LIN {X 0,Y 446.411,Z 696.876,A -85,B 0,C 180,E1 -8692.12,E2 -8692.12} C_VEL
LIN {X 0,Y 446.428,Z 696.878,A -85,B 0,C 180,E1 -8695.476,E2 -8695.476} C_VEL
LIN {X 0,Y 446.472,Z 697.063,A -85,B 0,C 180,E1 -8698.506,E2 -8698.506} C_VEL
LIN {X 0,Y 449.672,Z 710.867,A -85,B 0,C 180,E1 -8700.763,E2 -8700.763} C_VEL
LIN {X 0,Y 451.142,Z 718.019,A -85,B 0,C 180,E1 -8701.884,E2 -8701.884} C_VEL
LIN {X 0,Y 450.044,Z 738.904,A -85,B 0,C 180,E1 -8704.839,E2 -8704.839} C_VEL
LIN {X 0,Y 448.95,Z 761.08,A -85,B 0,C 180,E1 -8707.931,E2 -8707.931} C_VEL
LIN {X 0,Y 447.767,Z 788.534,A -85,B 0,C 180,E1 -8711.704,E2 -8711.704} C_VEL
LIN {X 0,Y 447.645,Z 792.086,A -85,B 0,C 180,E1 -8712.146,E2 -8712.146} C_VEL
LIN {X 0,Y 450.644,Z 820.359,A -85,B 0,C 180,E1 -8712.733,E2 -8712.733} C_VEL
LIN {X 0,Y 449.869,Z 902.501,A -85,B 0,C 180,E1 -8714.074,E2 -8714.074} C_VEL
LIN {X 0,Y 449.392,Z 915.74,A -85,B 0,C 180,E1 -8714.464,E2 -8714.464} C_VEL
LIN {X 0,Y 448.928,Z 927.38,A -85,B 0,C 180,E1 -8714.971,E2 -8714.971} C_VEL
LIN {X 0,Y 448.223,Z 939.892,A -85,B 0,C 180,E1 -8715.701,E2 -8715.701} C_VEL
LIN {X 0,Y 447.645,Z 951.783,A -85,B 0,C 180,E1 -8716.617,E2 -8716.617} C_VEL
LIN {X 0,Y 447.169,Z 962.339,A -85,B 0,C 180,E1 -8717.634,E2 -8717.634} C_VEL
LIN {X 0,Y 446.635,Z 971.045,A -85,B 0,C 180,E1 -8718.655,E2 -8718.655} C_VEL
LIN {X 0,Y 446.239,Z 979.102,A -85,B 0,C 180,E1 -8719.793,E2 -8719.793} C_VEL
LIN {X 0,Y 445.972,Z 987.009,A -85,B 0,C 180,E1 -8721.16,E2 -8721.16} C_VEL
LIN {X 0,Y 445.778,Z 994.294,A -85,B 0,C 180,E1 -8722.753,E2 -8722.753} C_VEL
LIN {X 0,Y 445.753,Z 999.161,A -85,B 0,C 180,E1 -8724.117,E2 -8724.117} C_VEL
LIN {X 0,Y 445.749,Z 1002.881,A -85,B 0,C 180,E1 -8725.477,E2 -8725.477} C_VEL
LIN {X 0,Y 445.775,Z 1004.802,A -85,B 0,C 180,E1 -8726.383,E2 -8726.383} C_VEL
LIN {X 0,Y 445.737,Z 1006.233,A -85,B 0,C 180,E1 -8727.287,E2 -8727.287} C_VEL
LIN {X 0,Y 445.739,Z 1007.252,A -85,B 0,C 180,E1 -8728.192,E2 -8728.192} C_VEL
LIN {X 0,Y 445.731,Z 1007.867,A -85,B 0,C 180,E1 -8729.095,E2 -8729.095} C_VEL
LIN {X 0,Y 445.738,Z 1008.078,A -85,B 0,C 180,E1 -8729.999,E2 -8729.999} C_VEL
LIN {X 0,Y 445.735,Z 1007.841,A -85,B 0,C 180,E1 -8730.902,E2 -8730.902} C_VEL
LIN {X 0,Y 445.746,Z 1007.198,A -85,B 0,C 180,E1 -8731.806,E2 -8731.806} C_VEL
LIN {X 0,Y 445.745,Z 1006.152,A -85,B 0,C 180,E1 -8732.71,E2 -8732.71} C_VEL
LIN {X 0,Y 445.774,Z 1004.693,A -85,B 0,C 180,E1 -8733.614,E2 -8733.614} C_VEL
LIN {X 0,Y 445.767,Z 1001.629,A -85,B 0,C 180,E1 -8734.973,E2 -8734.973} C_VEL
LIN {X 0,Y 445.748,Z 996.417,A -85,B 0,C 180,E1 -8736.632,E2 -8736.632} C_VEL
LIN {X 0,Y 445.887,Z 990.109,A -85,B 0,C 180,E1 -8738.154,E2 -8738.154} C_VEL
LIN {X 0,Y 446.086,Z 982.981,A -85,B 0,C 180,E1 -8739.521,E2 -8739.521} C_VEL
LIN {X 0,Y 446.484,Z 974.101,A -85,B 0,C 180,E1 -8740.887,E2 -8740.887} C_VEL
LIN {X 0,Y 446.893,Z 965.022,A -85,B 0,C 180,E1 -8742.026,E2 -8742.026} C_VEL
LIN {X 0,Y 447.39,Z 956.062,A -85,B 0,C 180,E1 -8742.956,E2 -8742.956} C_VEL
LIN {X 0,Y 447.891,Z 944.244,A -85,B 0,C 180,E1 -8743.959,E2 -8743.959} C_VEL
LIN {X 0,Y 448.619,Z 932.176,A -85,B 0,C 180,E1 -8744.747,E2 -8744.747} C_VEL
LIN {X 0,Y 449.176,Z 919.643,A -85,B 0,C 180,E1 -8745.366,E2 -8745.366} C_VEL
LIN {X 0,Y 449.722,Z 906.777,A -85,B 0,C 180,E1 -8745.812,E2 -8745.812} C_VEL
LIN {X 0,Y 449.986,Z 891.416,A -85,B 0,C 180,E1 -8746.122,E2 -8746.122} C_VEL
LIN {X 0,Y 450.614,Z 818.515,A -85,B 0,C 180,E1 -8747.294,E2 -8747.294} C_VEL
LIN {X 0,Y 447.578,Z 790.826,A -85,B 0,C 180,E1 -8747.892,E2 -8747.892} C_VEL
LIN {X 0,Y 448.442,Z 768.678,A -85,B 0,C 180,E1 -8750.886,E2 -8750.886} C_VEL
LIN {X 0,Y 449.417,Z 748.03,A -85,B 0,C 180,E1 -8753.744,E2 -8753.744} C_VEL
LIN {X 0,Y 450.55,Z 725.648,A -85,B 0,C 180,E1 -8756.894,E2 -8756.894} C_VEL
LIN {X 0,Y 450.925,Z 717.026,A -85,B 0,C 180,E1 -8758.128,E2 -8758.128} C_VEL
LIN {X 0,Y 447.652,Z 702.006,A -85,B 0,C 180,E1 -8760.532,E2 -8760.532} C_VEL
LIN {X 0,Y 446.437,Z 696.965,A -85,B 0,C 180,E1 -8761.428,E2 -8761.428} C_VEL
LIN {X 0,Y 446.423,Z 696.872,A -85,B 0,C 180,E1 -8764.522,E2 -8764.522} C_VEL
LIN {X 0,Y 446.409,Z 696.878,A -85,B 0,C 180,E1 -8768.078,E2 -8768.078} C_VEL
LIN {X 0,Y 446.42,Z 696.878,A -85,B 0,C 180,E1 -8770.916,E2 -8770.916} C_VEL
LIN {X 0,Y 446.394,Z 696.876,A -85,B 0,C 180,E1 -8773.845,E2 -8773.845} C_VEL
LIN {X 0,Y 446.415,Z 696.873,A -85,B 0,C 180,E1 -8776.399,E2 -8776.399} C_VEL
LIN {X 0,Y 446.439,Z 696.864,A -85,B 0,C 180,E1 -8779.802,E2 -8779.802} C_VEL
LIN {X 0,Y 446.418,Z 696.874,A -85,B 0,C 180,E1 -8782.122,E2 -8782.122} C_VEL
LIN {X 0,Y 446.421,Z 696.874,A -85,B 0,C 180,E1 -8785.476,E2 -8785.476} C_VEL
LIN {X 0,Y 446.409,Z 696.876,A -85,B 0,C 180,E1 -8788.699,E2 -8788.699} C_VEL
LIN {X 0,Y 446.473,Z 696.867,A -85,B 0,C 180,E1 -8791.821,E2 -8791.821} C_VEL
LIN {X 0,Y 446.447,Z 696.87,A -85,B 0,C 180,E1 -8794.847,E2 -8794.847} C_VEL
LIN {X 0,Y 446.436,Z 696.868,A -85,B 0,C 180,E1 -8798.244,E2 -8798.244} C_VEL
LIN {X 0,Y 446.446,Z 696.874,A -85,B 0,C 180,E1 -8801.649,E2 -8801.649} C_VEL
LIN {X 0,Y 446.504,Z 696.863,A -85,B 0,C 180,E1 -8804.48,E2 -8804.48} C_VEL
LIN {X 0,Y 446.505,Z 696.867,A -85,B 0,C 180,E1 -8808.193,E2 -8808.193} C_VEL
LIN {X 0,Y 446.588,Z 696.851,A -85,B 0,C 180,E1 -8811.858,E2 -8811.858} C_VEL
LIN {X 0,Y 446.63,Z 696.846,A -85,B 0,C 180,E1 -8814.583,E2 -8814.583} C_VEL
LIN {X 0,Y 446.698,Z 696.837,A -85,B 0,C 180,E1 -8817.295,E2 -8817.295} C_VEL
LIN {X 0,Y 446.78,Z 696.829,A -85,B 0,C 180,E1 -8820,E2 -8820} C_VEL
LIN {X 0,Y 446.696,Z 696.842,A -85,B 0,C 180,E1 -8822.706,E2 -8822.706} C_VEL
LIN {X 0,Y 446.627,Z 696.851,A -85,B 0,C 180,E1 -8826.324,E2 -8826.324} C_VEL
LIN {X 0,Y 446.527,Z 696.862,A -85,B 0,C 180,E1 -8829.056,E2 -8829.056} C_VEL
LIN {X 0,Y 446.509,Z 696.864,A -85,B 0,C 180,E1 -8832.73,E2 -8832.73} C_VEL
LIN {X 0,Y 446.484,Z 696.862,A -85,B 0,C 180,E1 -8836.228,E2 -8836.228} C_VEL
LIN {X 0,Y 446.457,Z 696.872,A -85,B 0,C 180,E1 -8839.304,E2 -8839.304} C_VEL
LIN {X 0,Y 446.406,Z 696.872,A -85,B 0,C 180,E1 -8842.2,E2 -8842.2} C_VEL
LIN {X 0,Y 446.428,Z 696.873,A -85,B 0,C 180,E1 -8845.154,E2 -8845.154} C_VEL
LIN {X 0,Y 446.475,Z 696.86,A -85,B 0,C 180,E1 -8848.18,E2 -8848.18} C_VEL
LIN {X 0,Y 446.41,Z 696.875,A -85,B 0,C 180,E1 -8851.776,E2 -8851.776} C_VEL
LIN {X 0,Y 446.421,Z 696.874,A -85,B 0,C 180,E1 -8854.524,E2 -8854.524} C_VEL
LIN {X 0,Y 446.422,Z 696.874,A -85,B 0,C 180,E1 -8858.083,E2 -8858.083} C_VEL
LIN {X 0,Y 446.419,Z 696.874,A -85,B 0,C 180,E1 -8860.919,E2 -8860.919} C_VEL
LIN {X 0,Y 446.393,Z 696.883,A -85,B 0,C 180,E1 -8863.847,E2 -8863.847} C_VEL
LIN {X 0,Y 446.424,Z 696.869,A -85,B 0,C 180,E1 -8866.781,E2 -8866.781} C_VEL
LIN {X 0,Y 446.468,Z 697.125,A -85,B 0,C 180,E1 -8867.456,E2 -8867.456} C_VEL
LIN {X 0,Y 446.776,Z 698.3,A -85,B 0,C 180,E1 -8867.596,E2 -8867.596} C_VEL
LIN {X 0,Y 451.11,Z 709.604,A -85,B 0,C 180,E1 -8867.983,E2 -8867.983} C_VEL
LIN {X 0,Y 450.672,Z 778.842,A -85,B 0,C 180,E1 -8869.143,E2 -8869.143} C_VEL
LIN {X 0,Y 450.538,Z 792.347,A -85,B 0,C 180,E1 -8869.566,E2 -8869.566} C_VEL
LIN {X 0,Y 450.352,Z 805.1,A -85,B 0,C 180,E1 -8870.162,E2 -8870.162} C_VEL
LIN {X 0,Y 450.013,Z 816.865,A -85,B 0,C 180,E1 -8870.911,E2 -8870.911} C_VEL
LIN {X 0,Y 449.474,Z 828.486,A -85,B 0,C 180,E1 -8871.859,E2 -8871.859} C_VEL
LIN {X 0,Y 448.979,Z 838.696,A -85,B 0,C 180,E1 -8872.914,E2 -8872.914} C_VEL
LIN {X 0,Y 448.445,Z 847.302,A -85,B 0,C 180,E1 -8874.008,E2 -8874.008} C_VEL
LIN {X 0,Y 447.898,Z 855.784,A -85,B 0,C 180,E1 -8875.335,E2 -8875.335} C_VEL
LIN {X 0,Y 447.493,Z 862.578,A -85,B 0,C 180,E1 -8876.657,E2 -8876.657} C_VEL
LIN {X 0,Y 447.072,Z 868.448,A -85,B 0,C 180,E1 -8878.091,E2 -8878.091} C_VEL
LIN {X 0,Y 446.774,Z 873.624,A -85,B 0,C 180,E1 -8879.778,E2 -8879.778} C_VEL
LIN {X 0,Y 446.617,Z 876.016,A -85,B 0,C 180,E1 -8880.805,E2 -8880.805} C_VEL
LIN {X 0,Y 446.483,Z 877.801,A -85,B 0,C 180,E1 -8881.823,E2 -8881.823} C_VEL
LIN {X 0,Y 446.403,Z 879.102,A -85,B 0,C 180,E1 -8882.836,E2 -8882.836} C_VEL
LIN {X 0,Y 446.335,Z 879.859,A -85,B 0,C 180,E1 -8883.841,E2 -8883.841} C_VEL
LIN {X 0,Y 446.292,Z 880.159,A -85,B 0,C 180,E1 -8884.839,E2 -8884.839} C_VEL
LIN {X 0,Y 446.282,Z 879.919,A -85,B 0,C 180,E1 -8885.977,E2 -8885.977} C_VEL
LIN {X 0,Y 446.374,Z 878.253,A -85,B 0,C 180,E1 -8887.8,E2 -8887.8} C_VEL
LIN {X 0,Y 446.558,Z 875.728,A -85,B 0,C 180,E1 -8889.263,E2 -8889.263} C_VEL
LIN {X 0,Y 446.761,Z 872.127,A -85,B 0,C 180,E1 -8890.712,E2 -8890.712} C_VEL
LIN {X 0,Y 446.814,Z 871.213,A -85,B 0,C 180,E1 -8891.008,E2 -8891.008} C_VEL
LIN {X 0,Y 446.302,Z 869.052,A -85,B 0,C 180,E1 -8891.709,E2 -8891.709} C_VEL
LIN {X 0,Y 443.732,Z 865.275,A -85,B 0,C 180,E1 -8892.844,E2 -8892.844} C_VEL
LIN {X 0,Y 441.198,Z 860.875,A -85,B 0,C 180,E1 -8893.948,E2 -8893.948} C_VEL
LIN {X 0,Y 440.742,Z 857.682,A -85,B 0,C 180,E1 -8894.594,E2 -8894.594} C_VEL
LIN {X 0,Y 441.292,Z 849.452,A -85,B 0,C 180,E1 -8895.945,E2 -8895.945} C_VEL
LIN {X 0,Y 441.805,Z 840.503,A -85,B 0,C 180,E1 -8897.134,E2 -8897.134} C_VEL
LIN {X 0,Y 442.34,Z 830.654,A -85,B 0,C 180,E1 -8898.198,E2 -8898.198} C_VEL
LIN {X 0,Y 442.866,Z 819.969,A -85,B 0,C 180,E1 -8899.129,E2 -8899.129} C_VEL
LIN {X 0,Y 443.254,Z 807.77,A -85,B 0,C 180,E1 -8899.957,E2 -8899.957} C_VEL
LIN {X 0,Y 443.562,Z 795.192,A -85,B 0,C 180,E1 -8900.597,E2 -8900.597} C_VEL
LIN {X 0,Y 443.715,Z 782.628,A -85,B 0,C 180,E1 -8901.044,E2 -8901.044} C_VEL
LIN {X 0,Y 443.753,Z 767.637,A -85,B 0,C 180,E1 -8901.355,E2 -8901.355} C_VEL
LIN {X 0,Y 444.215,Z 710.877,A -85,B 0,C 180,E1 -8902.29,E2 -8902.29} C_VEL
LIN {X 0,Y 439.707,Z 698.68,A -85,B 0,C 180,E1 -8902.707,E2 -8902.707} C_VEL
LIN {X 0,Y 439.558,Z 697.817,A -85,B 0,C 180,E1 -8902.883,E2 -8902.883} C_VEL
LIN {X 0,Y 439.599,Z 697.729,A -85,B 0,C 180,E1 -8904.497,E2 -8904.497} C_VEL
LIN {X 0,Y 439.629,Z 697.724,A -85,B 0,C 180,E1 -8908.169,E2 -8908.169} C_VEL
LIN {X 0,Y 439.672,Z 697.718,A -85,B 0,C 180,E1 -8910.001,E2 -8910.001} C_VEL
LIN {X 0,Y 439.605,Z 697.727,A -85,B 0,C 180,E1 -8912.75,E2 -8912.75} C_VEL
LIN {X 0,Y 439.562,Z 697.732,A -85,B 0,C 180,E1 -8916.427,E2 -8916.427} C_VEL
LIN {X 0,Y 439.476,Z 697.739,A -85,B 0,C 180,E1 -8919.203,E2 -8919.203} C_VEL
LIN {X 0,Y 439.47,Z 697.742,A -85,B 0,C 180,E1 -8922.939,E2 -8922.939} C_VEL
LIN {X 0,Y 439.45,Z 697.741,A -85,B 0,C 180,E1 -8926.348,E2 -8926.348} C_VEL
LIN {X 0,Y 439.385,Z 697.741,A -85,B 0,C 180,E1 -8929.628,E2 -8929.628} C_VEL
LIN {X 0,Y 439.367,Z 697.754,A -85,B 0,C 180,E1 -8932.577,E2 -8932.577} C_VEL
LIN {X 0,Y 439.349,Z 697.746,A -85,B 0,C 180,E1 -8935.59,E2 -8935.59} C_VEL
LIN {X 0,Y 439.383,Z 697.747,A -85,B 0,C 180,E1 -8938.677,E2 -8938.677} C_VEL
LIN {X 0,Y 439.348,Z 697.751,A -85,B 0,C 180,E1 -8942.025,E2 -8942.025} C_VEL
LIN {X 0,Y 439.388,Z 697.737,A -85,B 0,C 180,E1 -8945.338,E2 -8945.338} C_VEL
LIN {X 0,Y 439.353,Z 697.752,A -85,B 0,C 180,E1 -8948.599,E2 -8948.599} C_VEL
LIN {X 0,Y 439.35,Z 697.754,A -85,B 0,C 180,E1 -8952.211,E2 -8952.211} C_VEL
LIN {X 0,Y 439.377,Z 697.754,A -85,B 0,C 180,E1 -8955.267,E2 -8955.267} C_VEL
LIN {X 0,Y 439.365,Z 697.752,A -85,B 0,C 180,E1 -8958.748,E2 -8958.748} C_VEL
LIN {X 0,Y 439.355,Z 697.759,A -85,B 0,C 180,E1 -8961.613,E2 -8961.613} C_VEL
LIN {X 0,Y 439.357,Z 697.755,A -85,B 0,C 180,E1 -8964.84,E2 -8964.84} C_VEL
LIN {X 0,Y 439.352,Z 697.76,A -85,B 0,C 180,E1 -8968.137,E2 -8968.137} C_VEL
LIN {X 0,Y 439.423,Z 697.912,A -85,B 0,C 180,E1 -8969.481,E2 -8969.481} C_VEL
LIN {X 0,Y 439.563,Z 698.75,A -85,B 0,C 180,E1 -8969.623,E2 -8969.623} C_VEL
LIN {X 0,Y 443.704,Z 710.36,A -85,B 0,C 180,E1 -8970.015,E2 -8970.015} C_VEL
LIN {X 0,Y 443.036,Z 773.791,A -85,B 0,C 180,E1 -8971.157,E2 -8971.157} C_VEL
LIN {X 0,Y 442.834,Z 785.481,A -85,B 0,C 180,E1 -8971.507,E2 -8971.507} C_VEL
LIN {X 0,Y 442.604,Z 795.704,A -85,B 0,C 180,E1 -8971.939,E2 -8971.939} C_VEL
LIN {X 0,Y 442.436,Z 804.955,A -85,B 0,C 180,E1 -8972.442,E2 -8972.442} C_VEL
LIN {X 0,Y 441.975,Z 815.897,A -85,B 0,C 180,E1 -8973.193,E2 -8973.193} C_VEL
LIN {X 0,Y 441.652,Z 824.568,A -85,B 0,C 180,E1 -8973.922,E2 -8973.922} C_VEL
LIN {X 0,Y 441.184,Z 832.911,A -85,B 0,C 180,E1 -8974.754,E2 -8974.754} C_VEL
LIN {X 0,Y 440.818,Z 841.284,A -85,B 0,C 180,E1 -8975.761,E2 -8975.761} C_VEL
LIN {X 0,Y 440.485,Z 848.193,A -85,B 0,C 180,E1 -8976.741,E2 -8976.741} C_VEL
LIN {X 0,Y 440.108,Z 854.791,A -85,B 0,C 180,E1 -8977.851,E2 -8977.851} C_VEL
LIN {X 0,Y 439.75,Z 861.198,A -85,B 0,C 180,E1 -8979.17,E2 -8979.17} C_VEL
LIN {X 0,Y 439.507,Z 866.87,A -85,B 0,C 180,E1 -8980.642,E2 -8980.642} C_VEL
LIN {X 0,Y 439.289,Z 870.516,A -85,B 0,C 180,E1 -8981.822,E2 -8981.822} C_VEL
LIN {X 0,Y 439.14,Z 873.848,A -85,B 0,C 180,E1 -8983.257,E2 -8983.257} C_VEL
LIN {X 0,Y 439.079,Z 875.563,A -85,B 0,C 180,E1 -8984.21,E2 -8984.21} C_VEL
LIN {X 0,Y 439.007,Z 877.457,A -85,B 0,C 180,E1 -8986.105,E2 -8986.105} C_VEL
LIN {X 0,Y 439.052,Z 877.759,A -85,B 0,C 180,E1 -8987.542,E2 -8987.542} C_VEL
LIN {X 0,Y 439.106,Z 877.048,A -85,B 0,C 180,E1 -8988.927,E2 -8988.927} C_VEL
LIN {X 0,Y 439.205,Z 876.169,A -85,B 0,C 180,E1 -8989.862,E2 -8989.862} C_VEL
LIN {X 0,Y 439.405,Z 872.864,A -85,B 0,C 180,E1 -8991.723,E2 -8991.723} C_VEL
LIN {X 0,Y 439.571,Z 870.661,A -85,B 0,C 180,E1 -8992.651,E2 -8992.651} C_VEL
LIN {X 0,Y 439.83,Z 866.295,A -85,B 0,C 180,E1 -8994.038,E2 -8994.038} C_VEL
LIN {X 0,Y 440.123,Z 860.682,A -85,B 0,C 180,E1 -8995.42,E2 -8995.42} C_VEL
LIN {X 0,Y 440.456,Z 854.971,A -85,B 0,C 180,E1 -8996.569,E2 -8996.569} C_VEL
LIN {X 0,Y 440.907,Z 848.065,A -85,B 0,C 180,E1 -8997.716,E2 -8997.716} C_VEL
LIN {X 0,Y 441.349,Z 839.698,A -85,B 0,C 180,E1 -8998.859,E2 -8998.859} C_VEL
LIN {X 0,Y 441.764,Z 831.673,A -85,B 0,C 180,E1 -8999.772,E2 -8999.772} C_VEL
LIN {X 0,Y 442.208,Z 823.29,A -85,B 0,C 180,E1 -9000.569,E2 -9000.569} C_VEL
LIN {X 0,Y 442.55,Z 814.752,A -85,B 0,C 180,E1 -9001.251,E2 -9001.251} C_VEL
LIN {X 0,Y 442.87,Z 804.092,A -85,B 0,C 180,E1 -9001.932,E2 -9001.932} C_VEL
LIN {X 0,Y 443.183,Z 793.086,A -85,B 0,C 180,E1 -9002.471,E2 -9002.471} C_VEL
LIN {X 0,Y 443.272,Z 782.09,A -85,B 0,C 180,E1 -9002.868,E2 -9002.868} C_VEL
LIN {X 0,Y 443.347,Z 770.375,A -85,B 0,C 180,E1 -9003.152,E2 -9003.152} C_VEL
LIN {X 0,Y 444.19,Z 710.257,A -85,B 0,C 180,E1 -9004.252,E2 -9004.252} C_VEL
LIN {X 0,Y 439.633,Z 698.633,A -85,B 0,C 180,E1 -9004.728,E2 -9004.728} C_VEL
LIN {X 0,Y 439.496,Z 697.795,A -85,B 0,C 180,E1 -9004.931,E2 -9004.931} C_VEL
LIN {X 0,Y 439.56,Z 697.732,A -85,B 0,C 180,E1 -9007.556,E2 -9007.556} C_VEL
LIN {X 0,Y 439.467,Z 697.744,A -85,B 0,C 180,E1 -9010.132,E2 -9010.132} C_VEL
LIN {X 0,Y 439.473,Z 697.741,A -85,B 0,C 180,E1 -9012.937,E2 -9012.937} C_VEL
LIN {X 0,Y 439.454,Z 697.747,A -85,B 0,C 180,E1 -9016.348,E2 -9016.348} C_VEL
LIN {X 0,Y 439.409,Z 697.748,A -85,B 0,C 180,E1 -9019.626,E2 -9019.626} C_VEL
LIN {X 0,Y 439.371,Z 697.758,A -85,B 0,C 180,E1 -9022.575,E2 -9022.575} C_VEL
LIN {X 0,Y 439.387,Z 697.751,A -85,B 0,C 180,E1 -9025.586,E2 -9025.586} C_VEL
LIN {X 0,Y 439.407,Z 697.752,A -85,B 0,C 180,E1 -9028.674,E2 -9028.674} C_VEL
LIN {X 0,Y 439.375,Z 697.752,A -85,B 0,C 180,E1 -9032.029,E2 -9032.029} C_VEL
LIN {X 0,Y 439.399,Z 697.753,A -85,B 0,C 180,E1 -9035.339,E2 -9035.339} C_VEL
LIN {X 0,Y 439.39,Z 697.752,A -85,B 0,C 180,E1 -9038.594,E2 -9038.594} C_VEL
LIN {X 0,Y 439.395,Z 697.753,A -85,B 0,C 180,E1 -9041.256,E2 -9041.256} C_VEL
LIN {X 0,Y 439.406,Z 697.75,A -85,B 0,C 180,E1 -9044.729,E2 -9044.729} C_VEL
LIN {X 0,Y 439.402,Z 697.752,A -85,B 0,C 180,E1 -9047.795,E2 -9047.795} C_VEL
LIN {X 0,Y 439.395,Z 697.749,A -85,B 0,C 180,E1 -9050.222,E2 -9050.222} C_VEL
LIN {X 0,Y 439.377,Z 697.756,A -85,B 0,C 180,E1 -9053.712,E2 -9053.712} C_VEL
LIN {X 0,Y 439.377,Z 697.755,A -85,B 0,C 180,E1 -9057.053,E2 -9057.053} C_VEL
LIN {X 0,Y 439.432,Z 698.009,A -85,B 0,C 180,E1 -9058.244,E2 -9058.244} C_VEL
LIN {X 0,Y 442.655,Z 711.641,A -85,B 0,C 180,E1 -9060.514,E2 -9060.514} C_VEL
LIN {X 0,Y 444.151,Z 718.815,A -85,B 0,C 180,E1 -9061.659,E2 -9061.659} C_VEL
LIN {X 0,Y 444.197,Z 722.176,A -85,B 0,C 180,E1 -9062.158,E2 -9062.158} C_VEL
LIN {X 0,Y 442.914,Z 742.94,A -85,B 0,C 180,E1 -9065.135,E2 -9065.135} C_VEL
LIN {X 0,Y 441.853,Z 763.539,A -85,B 0,C 180,E1 -9068.049,E2 -9068.049} C_VEL
LIN {X 0,Y 440.712,Z 789.399,A -85,B 0,C 180,E1 -9071.665,E2 -9071.665} C_VEL
LIN {X 0,Y 440.678,Z 790.898,A -85,B 0,C 180,E1 -9071.849,E2 -9071.849} C_VEL
LIN {X 0,Y 443.816,Z 820.934,A -85,B 0,C 180,E1 -9072.489,E2 -9072.489} C_VEL
LIN {X 0,Y 443.053,Z 901.376,A -85,B 0,C 180,E1 -9073.823,E2 -9073.823} C_VEL
LIN {X 0,Y 442.51,Z 914.65,A -85,B 0,C 180,E1 -9074.217,E2 -9074.217} C_VEL
LIN {X 0,Y 441.975,Z 927.448,A -85,B 0,C 180,E1 -9074.788,E2 -9074.788} C_VEL
LIN {X 0,Y 441.297,Z 938.844,A -85,B 0,C 180,E1 -9075.472,E2 -9075.472} C_VEL
LIN {X 0,Y 440.68,Z 950.445,A -85,B 0,C 180,E1 -9076.375,E2 -9076.375} C_VEL
LIN {X 0,Y 440.189,Z 961.306,A -85,B 0,C 180,E1 -9077.434,E2 -9077.434} C_VEL
LIN {X 0,Y 439.605,Z 970.012,A -85,B 0,C 180,E1 -9078.471,E2 -9078.471} C_VEL
LIN {X 0,Y 439.208,Z 978.077,A -85,B 0,C 180,E1 -9079.628,E2 -9079.628} C_VEL
LIN {X 0,Y 438.894,Z 985.985,A -85,B 0,C 180,E1 -9081.017,E2 -9081.017} C_VEL
LIN {X 0,Y 438.735,Z 993.279,A -85,B 0,C 180,E1 -9082.636,E2 -9082.636} C_VEL
LIN {X 0,Y 438.695,Z 998.148,A -85,B 0,C 180,E1 -9084.022,E2 -9084.022} C_VEL
LIN {X 0,Y 438.709,Z 1001.873,A -85,B 0,C 180,E1 -9085.404,E2 -9085.404} C_VEL
LIN {X 0,Y 438.736,Z 1003.795,A -85,B 0,C 180,E1 -9086.325,E2 -9086.325} C_VEL
LIN {X 0,Y 438.697,Z 1005.228,A -85,B 0,C 180,E1 -9087.244,E2 -9087.244} C_VEL
LIN {X 0,Y 438.702,Z 1006.247,A -85,B 0,C 180,E1 -9088.163,E2 -9088.163} C_VEL
LIN {X 0,Y 438.7,Z 1006.861,A -85,B 0,C 180,E1 -9089.081,E2 -9089.081} C_VEL
LIN {X 0,Y 438.71,Z 1007.072,A -85,B 0,C 180,E1 -9089.999,E2 -9089.999} C_VEL
LIN {X 0,Y 438.704,Z 1006.833,A -85,B 0,C 180,E1 -9090.917,E2 -9090.917} C_VEL
LIN {X 0,Y 438.71,Z 1006.188,A -85,B 0,C 180,E1 -9091.835,E2 -9091.835} C_VEL
LIN {X 0,Y 438.704,Z 1005.138,A -85,B 0,C 180,E1 -9092.753,E2 -9092.753} C_VEL
LIN {X 0,Y 438.736,Z 1003.677,A -85,B 0,C 180,E1 -9093.672,E2 -9093.672} C_VEL
LIN {X 0,Y 438.723,Z 1000.607,A -85,B 0,C 180,E1 -9095.053,E2 -9095.053} C_VEL
LIN {X 0,Y 438.684,Z 995.728,A -85,B 0,C 180,E1 -9096.645,E2 -9096.645} C_VEL
LIN {X 0,Y 438.849,Z 989.073,A -85,B 0,C 180,E1 -9098.286,E2 -9098.286} C_VEL
LIN {X 0,Y 439.036,Z 981.936,A -85,B 0,C 180,E1 -9099.675,E2 -9099.675} C_VEL
LIN {X 0,Y 439.426,Z 973.047,A -85,B 0,C 180,E1 -9101.064,E2 -9101.064} C_VEL
LIN {X 0,Y 439.922,Z 963.973,A -85,B 0,C 180,E1 -9102.219,E2 -9102.219} C_VEL
LIN {X 0,Y 440.479,Z 953.239,A -85,B 0,C 180,E1 -9103.336,E2 -9103.336} C_VEL
LIN {X 0,Y 441.036,Z 941.614,A -85,B 0,C 180,E1 -9104.298,E2 -9104.298} C_VEL
LIN {X 0,Y 441.86,Z 929.134,A -85,B 0,C 180,E1 -9105.095,E2 -9105.095} C_VEL
LIN {X 0,Y 442.377,Z 917.318,A -85,B 0,C 180,E1 -9105.667,E2 -9105.667} C_VEL
LIN {X 0,Y 442.872,Z 904.71,A -85,B 0,C 180,E1 -9106.092,E2 -9106.092} C_VEL
LIN {X 0,Y 443.154,Z 888.772,A -85,B 0,C 180,E1 -9106.407,E2 -9106.407} C_VEL
LIN {X 0,Y 443.713,Z 818.543,A -85,B 0,C 180,E1 -9107.559,E2 -9107.559} C_VEL
LIN {X 0,Y 440.628,Z 789.544,A -85,B 0,C 180,E1 -9108.204,E2 -9108.204} C_VEL
LIN {X 0,Y 441.791,Z 762.525,A -85,B 0,C 180,E1 -9111.951,E2 -9111.951} C_VEL
LIN {X 0,Y 442.938,Z 740.095,A -85,B 0,C 180,E1 -9115.13,E2 -9115.13} C_VEL
LIN {X 0,Y 444.111,Z 719.45,A -85,B 0,C 180,E1 -9118.107,E2 -9118.107} C_VEL
LIN {X 0,Y 441.632,Z 707.191,A -85,B 0,C 180,E1 -9120.083,E2 -9120.083} C_VEL
LIN {X 0,Y 439.387,Z 697.884,A -85,B 0,C 180,E1 -9121.689,E2 -9121.689} C_VEL
LIN {X 0,Y 439.381,Z 697.746,A -85,B 0,C 180,E1 -9124.042,E2 -9124.042} C_VEL
LIN {X 0,Y 439.342,Z 697.761,A -85,B 0,C 180,E1 -9126.886,E2 -9126.886} C_VEL
LIN {X 0,Y 439.394,Z 697.751,A -85,B 0,C 180,E1 -9129.848,E2 -9129.848} C_VEL
LIN {X 0,Y 439.374,Z 697.753,A -85,B 0,C 180,E1 -9132.626,E2 -9132.626} C_VEL
LIN {X 0,Y 439.398,Z 697.748,A -85,B 0,C 180,E1 -9135.27,E2 -9135.27} C_VEL
LIN {X 0,Y 439.381,Z 697.755,A -85,B 0,C 180,E1 -9138.742,E2 -9138.742} C_VEL
LIN {X 0,Y 439.375,Z 697.753,A -85,B 0,C 180,E1 -9141.605,E2 -9141.605} C_VEL
LIN {X 0,Y 439.391,Z 697.744,A -85,B 0,C 180,E1 -9144.843,E2 -9144.843} C_VEL
LIN {X 0,Y 439.364,Z 697.752,A -85,B 0,C 180,E1 -9148.139,E2 -9148.139} C_VEL
LIN {X 0,Y 439.414,Z 697.75,A -85,B 0,C 180,E1 -9151.326,E2 -9151.326} C_VEL
LIN {X 0,Y 439.394,Z 697.747,A -85,B 0,C 180,E1 -9154.414,E2 -9154.414} C_VEL
LIN {X 0,Y 439.354,Z 697.76,A -85,B 0,C 180,E1 -9157.424,E2 -9157.424} C_VEL
LIN {X 0,Y 439.429,Z 697.744,A -85,B 0,C 180,E1 -9160.662,E2 -9160.662} C_VEL
LIN {X 0,Y 439.463,Z 697.742,A -85,B 0,C 180,E1 -9164.225,E2 -9164.225} C_VEL
LIN {X 0,Y 439.471,Z 697.744,A -85,B 0,C 180,E1 -9168.001,E2 -9168.001} C_VEL
LIN {X 0,Y 439.536,Z 697.728,A -85,B 0,C 180,E1 -9171.726,E2 -9171.726} C_VEL
LIN {X 0,Y 439.605,Z 697.722,A -85,B 0,C 180,E1 -9174.496,E2 -9174.496} C_VEL
LIN {X 0,Y 439.624,Z 697.725,A -85,B 0,C 180,E1 -9178.168,E2 -9178.168} C_VEL
LIN {X 0,Y 439.751,Z 697.705,A -85,B 0,C 180,E1 -9180,E2 -9180} C_VEL
LIN {X 0,Y 439.643,Z 697.72,A -85,B 0,C 180,E1 -9182.749,E2 -9182.749} C_VEL
LIN {X 0,Y 439.601,Z 697.727,A -85,B 0,C 180,E1 -9186.426,E2 -9186.426} C_VEL
LIN {X 0,Y 439.489,Z 697.738,A -85,B 0,C 180,E1 -9189.202,E2 -9189.202} C_VEL
LIN {X 0,Y 439.453,Z 697.744,A -85,B 0,C 180,E1 -9192.938,E2 -9192.938} C_VEL
LIN {X 0,Y 439.435,Z 697.741,A -85,B 0,C 180,E1 -9196.349,E2 -9196.349} C_VEL
LIN {X 0,Y 439.391,Z 697.75,A -85,B 0,C 180,E1 -9199.627,E2 -9199.627} C_VEL
LIN {X 0,Y 439.352,Z 697.752,A -85,B 0,C 180,E1 -9202.576,E2 -9202.576} C_VEL
LIN {X 0,Y 439.377,Z 697.757,A -85,B 0,C 180,E1 -9205.587,E2 -9205.587} C_VEL
LIN {X 0,Y 439.407,Z 697.74,A -85,B 0,C 180,E1 -9208.675,E2 -9208.675} C_VEL
LIN {X 0,Y 439.361,Z 697.75,A -85,B 0,C 180,E1 -9212.032,E2 -9212.032} C_VEL
LIN {X 0,Y 439.387,Z 697.753,A -85,B 0,C 180,E1 -9215.342,E2 -9215.342} C_VEL
LIN {X 0,Y 439.382,Z 697.747,A -85,B 0,C 180,E1 -9218.596,E2 -9218.596} C_VEL
LIN {X 0,Y 439.381,Z 697.751,A -85,B 0,C 180,E1 -9221.258,E2 -9221.258} C_VEL
LIN {X 0,Y 439.392,Z 697.752,A -85,B 0,C 180,E1 -9224.731,E2 -9224.731} C_VEL
LIN {X 0,Y 439.396,Z 697.855,A -85,B 0,C 180,E1 -9227.096,E2 -9227.096} C_VEL
LIN {X 0,Y 439.574,Z 698.672,A -85,B 0,C 180,E1 -9227.262,E2 -9227.262} C_VEL
LIN {X 0,Y 444.534,Z 711.592,A -85,B 0,C 180,E1 -9227.732,E2 -9227.732} C_VEL
LIN {X 0,Y 443.906,Z 779.538,A -85,B 0,C 180,E1 -9228.882,E2 -9228.882} C_VEL
LIN {X 0,Y 443.782,Z 792.792,A -85,B 0,C 180,E1 -9229.297,E2 -9229.297} C_VEL
LIN {X 0,Y 443.601,Z 805.01,A -85,B 0,C 180,E1 -9229.865,E2 -9229.865} C_VEL
LIN {X 0,Y 443.328,Z 815.314,A -85,B 0,C 180,E1 -9230.501,E2 -9230.501} C_VEL
LIN {X 0,Y 442.818,Z 826.743,A -85,B 0,C 180,E1 -9231.397,E2 -9231.397} C_VEL
LIN {X 0,Y 442.311,Z 836.551,A -85,B 0,C 180,E1 -9232.363,E2 -9232.363} C_VEL
LIN {X 0,Y 441.719,Z 846.051,A -85,B 0,C 180,E1 -9233.514,E2 -9233.514} C_VEL
LIN {X 0,Y 441.143,Z 854.523,A -85,B 0,C 180,E1 -9234.778,E2 -9234.778} C_VEL
LIN {X 0,Y 440.687,Z 861.508,A -85,B 0,C 180,E1 -9236.072,E2 -9236.072} C_VEL
LIN {X 0,Y 440.26,Z 867.787,A -85,B 0,C 180,E1 -9237.526,E2 -9237.526} C_VEL
LIN {X 0,Y 439.84,Z 873.504,A -85,B 0,C 180,E1 -9239.25,E2 -9239.25} C_VEL
LIN {X 0,Y 439.607,Z 877.196,A -85,B 0,C 180,E1 -9240.819,E2 -9240.819} C_VEL
LIN {X 0,Y 439.431,Z 879.627,A -85,B 0,C 180,E1 -9242.369,E2 -9242.369} C_VEL
LIN {X 0,Y 439.344,Z 880.774,A -85,B 0,C 180,E1 -9243.613,E2 -9243.613} C_VEL
LIN {X 0,Y 439.265,Z 881.117,A -85,B 0,C 180,E1 -9245.42,E2 -9245.42} C_VEL
LIN {X 0,Y 439.258,Z 880.689,A -85,B 0,C 180,E1 -9246.424,E2 -9246.424} C_VEL
LIN {X 0,Y 439.393,Z 878.918,A -85,B 0,C 180,E1 -9248.08,E2 -9248.08} C_VEL
LIN {X 0,Y 439.639,Z 875.436,A -85,B 0,C 180,E1 -9249.899,E2 -9249.899} C_VEL
LIN {X 0,Y 439.881,Z 871.384,A -85,B 0,C 180,E1 -9251.366,E2 -9251.366} C_VEL
LIN {X 0,Y 440.237,Z 866.1,A -85,B 0,C 180,E1 -9252.824,E2 -9252.824} C_VEL
LIN {X 0,Y 440.64,Z 859.405,A -85,B 0,C 180,E1 -9254.269,E2 -9254.269} C_VEL
LIN {X 0,Y 440.742,Z 857.682,A -85,B 0,C 180,E1 -9254.594,E2 -9254.594} C_VEL
LIN {X 0,Y 440.292,Z 854.298,A -85,B 0,C 180,E1 -9255.224,E2 -9255.224} C_VEL
LIN {X 0,Y 437.825,Z 848.624,A -85,B 0,C 180,E1 -9256.241,E2 -9256.241} C_VEL
LIN {X 0,Y 435.444,Z 842.352,A -85,B 0,C 180,E1 -9257.198,E2 -9257.198} C_VEL
LIN {X 0,Y 435.117,Z 838.04,A -85,B 0,C 180,E1 -9257.725,E2 -9257.725} C_VEL
LIN {X 0,Y 435.696,Z 826.957,A -85,B 0,C 180,E1 -9258.841,E2 -9258.841} C_VEL
LIN {X 0,Y 436.214,Z 816.56,A -85,B 0,C 180,E1 -9259.674,E2 -9259.674} C_VEL
LIN {X 0,Y 436.576,Z 804.208,A -85,B 0,C 180,E1 -9260.446,E2 -9260.446} C_VEL
LIN {X 0,Y 436.822,Z 791.29,A -85,B 0,C 180,E1 -9261.035,E2 -9261.035} C_VEL
LIN {X 0,Y 436.958,Z 778.781,A -85,B 0,C 180,E1 -9261.416,E2 -9261.416} C_VEL
LIN {X 0,Y 437.466,Z 712.472,A -85,B 0,C 180,E1 -9262.544,E2 -9262.544} C_VEL
LIN {X 0,Y 432.708,Z 699.615,A -85,B 0,C 180,E1 -9262.992,E2 -9262.992} C_VEL
LIN {X 0,Y 432.533,Z 698.685,A -85,B 0,C 180,E1 -9263.184,E2 -9263.184} C_VEL
LIN {X 0,Y 432.574,Z 698.605,A -85,B 0,C 180,E1 -9264.407,E2 -9264.407} C_VEL
LIN {X 0,Y 432.599,Z 698.599,A -85,B 0,C 180,E1 -9268.139,E2 -9268.139} C_VEL
LIN {X 0,Y 432.623,Z 698.595,A -85,B 0,C 180,E1 -9270.001,E2 -9270.001} C_VEL
LIN {X 0,Y 432.558,Z 698.605,A -85,B 0,C 180,E1 -9272.795,E2 -9272.795} C_VEL
LIN {X 0,Y 432.519,Z 698.608,A -85,B 0,C 180,E1 -9276.532,E2 -9276.532} C_VEL
LIN {X 0,Y 432.422,Z 698.617,A -85,B 0,C 180,E1 -9279.355,E2 -9279.355} C_VEL
LIN {X 0,Y 432.436,Z 698.62,A -85,B 0,C 180,E1 -9282.804,E2 -9282.804} C_VEL
LIN {X 0,Y 432.416,Z 698.619,A -85,B 0,C 180,E1 -9286.478,E2 -9286.478} C_VEL
LIN {X 0,Y 432.322,Z 698.62,A -85,B 0,C 180,E1 -9289.963,E2 -9289.963} C_VEL
LIN {X 0,Y 432.315,Z 698.638,A -85,B 0,C 180,E1 -9292.966,E2 -9292.966} C_VEL
LIN {X 0,Y 432.301,Z 698.622,A -85,B 0,C 180,E1 -9296.038,E2 -9296.038} C_VEL
LIN {X 0,Y 432.321,Z 698.633,A -85,B 0,C 180,E1 -9299.19,E2 -9299.19} C_VEL
LIN {X 0,Y 432.311,Z 698.628,A -85,B 0,C 180,E1 -9302.445,E2 -9302.445} C_VEL
LIN {X 0,Y 432.336,Z 698.62,A -85,B 0,C 180,E1 -9305.819,E2 -9305.819} C_VEL
LIN {X 0,Y 432.317,Z 698.629,A -85,B 0,C 180,E1 -9308.71,E2 -9308.71} C_VEL
LIN {X 0,Y 432.306,Z 698.636,A -85,B 0,C 180,E1 -9311.802,E2 -9311.802} C_VEL
LIN {X 0,Y 432.317,Z 698.63,A -85,B 0,C 180,E1 -9314.351,E2 -9314.351} C_VEL
LIN {X 0,Y 432.306,Z 698.632,A -85,B 0,C 180,E1 -9317.019,E2 -9317.019} C_VEL
LIN {X 0,Y 432.294,Z 698.639,A -85,B 0,C 180,E1 -9319.829,E2 -9319.829} C_VEL
LIN {X 0,Y 432.293,Z 698.634,A -85,B 0,C 180,E1 -9323.02,E2 -9323.02} C_VEL
LIN {X 0,Y 432.327,Z 698.635,A -85,B 0,C 180,E1 -9326.005,E2 -9326.005} C_VEL
LIN {X 0,Y 432.377,Z 698.802,A -85,B 0,C 180,E1 -9329.229,E2 -9329.229} C_VEL
LIN {X 0,Y 432.617,Z 699.893,A -85,B 0,C 180,E1 -9329.387,E2 -9329.387} C_VEL
LIN {X 0,Y 436.893,Z 712.016,A -85,B 0,C 180,E1 -9329.79,E2 -9329.79} C_VEL
LIN {X 0,Y 436.19,Z 774.897,A -85,B 0,C 180,E1 -9330.946,E2 -9330.946} C_VEL
LIN {X 0,Y 435.974,Z 786.708,A -85,B 0,C 180,E1 -9331.309,E2 -9331.309} C_VEL
LIN {X 0,Y 435.73,Z 797.544,A -85,B 0,C 180,E1 -9331.784,E2 -9331.784} C_VEL
LIN {X 0,Y 435.517,Z 806.462,A -85,B 0,C 180,E1 -9332.284,E2 -9332.284} C_VEL
LIN {X 0,Y 435.1,Z 816.365,A -85,B 0,C 180,E1 -9332.971,E2 -9332.971} C_VEL
LIN {X 0,Y 434.739,Z 825.355,A -85,B 0,C 180,E1 -9333.733,E2 -9333.733} C_VEL
LIN {X 0,Y 434.232,Z 834.363,A -85,B 0,C 180,E1 -9334.653,E2 -9334.653} C_VEL
LIN {X 0,Y 433.881,Z 842.148,A -85,B 0,C 180,E1 -9335.603,E2 -9335.603} C_VEL
LIN {X 0,Y 433.542,Z 849.089,A -85,B 0,C 180,E1 -9336.599,E2 -9336.599} C_VEL
LIN {X 0,Y 433.119,Z 855.956,A -85,B 0,C 180,E1 -9337.775,E2 -9337.775} C_VEL
LIN {X 0,Y 432.782,Z 862.146,A -85,B 0,C 180,E1 -9339.068,E2 -9339.068} C_VEL
LIN {X 0,Y 432.516,Z 867.542,A -85,B 0,C 180,E1 -9340.47,E2 -9340.47} C_VEL
LIN {X 0,Y 432.338,Z 870.9,A -85,B 0,C 180,E1 -9341.519,E2 -9341.519} C_VEL
LIN {X 0,Y 432.148,Z 874.429,A -85,B 0,C 180,E1 -9342.978,E2 -9342.978} C_VEL
LIN {X 0,Y 432.097,Z 876.17,A -85,B 0,C 180,E1 -9343.948,E2 -9343.948} C_VEL
LIN {X 0,Y 431.999,Z 878.347,A -85,B 0,C 180,E1 -9345.875,E2 -9345.875} C_VEL
LIN {X 0,Y 432.042,Z 878.812,A -85,B 0,C 180,E1 -9347.43,E2 -9347.43} C_VEL
LIN {X 0,Y 432.085,Z 878.311,A -85,B 0,C 180,E1 -9348.744,E2 -9348.744} C_VEL
LIN {X 0,Y 432.165,Z 877.455,A -85,B 0,C 180,E1 -9349.695,E2 -9349.695} C_VEL
LIN {X 0,Y 432.414,Z 874.445,A -85,B 0,C 180,E1 -9351.589,E2 -9351.589} C_VEL
LIN {X 0,Y 432.68,Z 870.993,A -85,B 0,C 180,E1 -9353.003,E2 -9353.003} C_VEL
LIN {X 0,Y 432.917,Z 866.439,A -85,B 0,C 180,E1 -9354.41,E2 -9354.41} C_VEL
LIN {X 0,Y 433.192,Z 861.729,A -85,B 0,C 180,E1 -9355.58,E2 -9355.58} C_VEL
LIN {X 0,Y 433.587,Z 856.003,A -85,B 0,C 180,E1 -9356.748,E2 -9356.748} C_VEL
LIN {X 0,Y 434.059,Z 849.077,A -85,B 0,C 180,E1 -9357.912,E2 -9357.912} C_VEL
LIN {X 0,Y 434.531,Z 840.68,A -85,B 0,C 180,E1 -9359.073,E2 -9359.073} C_VEL
LIN {X 0,Y 434.96,Z 832.623,A -85,B 0,C 180,E1 -9360,E2 -9360} C_VEL
LIN {X 0,Y 435.428,Z 824.193,A -85,B 0,C 180,E1 -9360.809,E2 -9360.809} C_VEL
LIN {X 0,Y 435.785,Z 815.595,A -85,B 0,C 180,E1 -9361.502,E2 -9361.502} C_VEL
LIN {X 0,Y 436.11,Z 804.646,A -85,B 0,C 180,E1 -9362.205,E2 -9362.205} C_VEL
LIN {X 0,Y 436.421,Z 793.756,A -85,B 0,C 180,E1 -9362.74,E2 -9362.74} C_VEL
LIN {X 0,Y 436.523,Z 783.035,A -85,B 0,C 180,E1 -9363.131,E2 -9363.131} C_VEL
LIN {X 0,Y 436.583,Z 770.094,A -85,B 0,C 180,E1 -9363.444,E2 -9363.444} C_VEL
LIN {X 0,Y 437.434,Z 711.704,A -85,B 0,C 180,E1 -9364.544,E2 -9364.544} C_VEL
LIN {X 0,Y 432.659,Z 699.544,A -85,B 0,C 180,E1 -9365.061,E2 -9365.061} C_VEL
LIN {X 0,Y 432.519,Z 698.696,A -85,B 0,C 180,E1 -9365.244,E2 -9365.244} C_VEL
LIN {X 0,Y 432.521,Z 698.609,A -85,B 0,C 180,E1 -9367.606,E2 -9367.606} C_VEL
LIN {X 0,Y 432.412,Z 698.623,A -85,B 0,C 180,E1 -9370.299,E2 -9370.299} C_VEL
LIN {X 0,Y 432.408,Z 698.62,A -85,B 0,C 180,E1 -9373.152,E2 -9373.152} C_VEL
LIN {X 0,Y 432.419,Z 698.623,A -85,B 0,C 180,E1 -9376.478,E2 -9376.478} C_VEL
LIN {X 0,Y 432.346,Z 698.63,A -85,B 0,C 180,E1 -9379.96,E2 -9379.96} C_VEL
LIN {X 0,Y 432.325,Z 698.632,A -85,B 0,C 180,E1 -9382.964,E2 -9382.964} C_VEL
LIN {X 0,Y 432.346,Z 698.63,A -85,B 0,C 180,E1 -9385.002,E2 -9385.002} C_VEL
LIN {X 0,Y 432.354,Z 698.628,A -85,B 0,C 180,E1 -9388.125,E2 -9388.125} C_VEL
LIN {X 0,Y 432.327,Z 698.632,A -85,B 0,C 180,E1 -9391.346,E2 -9391.346} C_VEL
LIN {X 0,Y 432.344,Z 698.63,A -85,B 0,C 180,E1 -9394.677,E2 -9394.677} C_VEL
LIN {X 0,Y 432.345,Z 698.628,A -85,B 0,C 180,E1 -9398.149,E2 -9398.149} C_VEL
LIN {X 0,Y 432.339,Z 698.632,A -85,B 0,C 180,E1 -9401.601,E2 -9401.601} C_VEL
LIN {X 0,Y 432.34,Z 698.629,A -85,B 0,C 180,E1 -9404.347,E2 -9404.347} C_VEL
LIN {X 0,Y 432.326,Z 698.633,A -85,B 0,C 180,E1 -9407.015,E2 -9407.015} C_VEL
LIN {X 0,Y 432.34,Z 698.631,A -85,B 0,C 180,E1 -9409.82,E2 -9409.82} C_VEL
LIN {X 0,Y 432.31,Z 698.633,A -85,B 0,C 180,E1 -9413.021,E2 -9413.021} C_VEL
LIN {X 0,Y 432.363,Z 698.629,A -85,B 0,C 180,E1 -9415.996,E2 -9415.996} C_VEL
LIN {X 0,Y 432.358,Z 698.811,A -85,B 0,C 180,E1 -9417.937,E2 -9417.937} C_VEL
LIN {X 0,Y 435.706,Z 712.921,A -85,B 0,C 180,E1 -9420.336,E2 -9420.336} C_VEL
LIN {X 0,Y 437.361,Z 721.35,A -85,B 0,C 180,E1 -9421.702,E2 -9421.702} C_VEL
LIN {X 0,Y 436.042,Z 742.624,A -85,B 0,C 180,E1 -9424.807,E2 -9424.807} C_VEL
LIN {X 0,Y 434.96,Z 762.558,A -85,B 0,C 180,E1 -9427.683,E2 -9427.683} C_VEL
LIN {X 0,Y 433.691,Z 789.373,A -85,B 0,C 180,E1 -9431.492,E2 -9431.492} C_VEL
LIN {X 0,Y 433.776,Z 790.824,A -85,B 0,C 180,E1 -9431.581,E2 -9431.581} C_VEL
LIN {X 0,Y 437.006,Z 820.85,A -85,B 0,C 180,E1 -9432.228,E2 -9432.228} C_VEL
LIN {X 0,Y 436.182,Z 901.238,A -85,B 0,C 180,E1 -9433.591,E2 -9433.591} C_VEL
LIN {X 0,Y 435.59,Z 915,A -85,B 0,C 180,E1 -9434.019,E2 -9434.019} C_VEL
LIN {X 0,Y 435.032,Z 927.431,A -85,B 0,C 180,E1 -9434.599,E2 -9434.599} C_VEL
LIN {X 0,Y 434.275,Z 939.365,A -85,B 0,C 180,E1 -9435.352,E2 -9435.352} C_VEL
LIN {X 0,Y 433.642,Z 950.773,A -85,B 0,C 180,E1 -9436.276,E2 -9436.276} C_VEL
LIN {X 0,Y 433.145,Z 961.344,A -85,B 0,C 180,E1 -9437.346,E2 -9437.346} C_VEL
LIN {X 0,Y 432.497,Z 970.716,A -85,B 0,C 180,E1 -9438.517,E2 -9438.517} C_VEL
LIN {X 0,Y 432.016,Z 979.86,A -85,B 0,C 180,E1 -9439.927,E2 -9439.927} C_VEL
LIN {X 0,Y 431.797,Z 987.26,A -85,B 0,C 180,E1 -9441.34,E2 -9441.34} C_VEL
LIN {X 0,Y 431.656,Z 992.26,A -85,B 0,C 180,E1 -9442.515,E2 -9442.515} C_VEL
LIN {X 0,Y 431.639,Z 997.135,A -85,B 0,C 180,E1 -9443.923,E2 -9443.923} C_VEL
LIN {X 0,Y 431.666,Z 1000.865,A -85,B 0,C 180,E1 -9445.329,E2 -9445.329} C_VEL
LIN {X 0,Y 431.699,Z 1002.789,A -85,B 0,C 180,E1 -9446.265,E2 -9446.265} C_VEL
LIN {X 0,Y 431.656,Z 1004.222,A -85,B 0,C 180,E1 -9447.199,E2 -9447.199} C_VEL
LIN {X 0,Y 431.665,Z 1005.241,A -85,B 0,C 180,E1 -9448.133,E2 -9448.133} C_VEL
LIN {X 0,Y 431.669,Z 1005.855,A -85,B 0,C 180,E1 -9449.066,E2 -9449.066} C_VEL
LIN {X 0,Y 431.681,Z 1006.065,A -85,B 0,C 180,E1 -9449.999,E2 -9449.999} C_VEL
LIN {X 0,Y 431.673,Z 1005.826,A -85,B 0,C 180,E1 -9450.931,E2 -9450.931} C_VEL
LIN {X 0,Y 431.673,Z 1005.177,A -85,B 0,C 180,E1 -9451.865,E2 -9451.865} C_VEL
LIN {X 0,Y 431.664,Z 1004.124,A -85,B 0,C 180,E1 -9452.798,E2 -9452.798} C_VEL
LIN {X 0,Y 431.699,Z 1002.661,A -85,B 0,C 180,E1 -9453.732,E2 -9453.732} C_VEL
LIN {X 0,Y 431.658,Z 999.582,A -85,B 0,C 180,E1 -9455.136,E2 -9455.136} C_VEL
LIN {X 0,Y 431.613,Z 995.07,A -85,B 0,C 180,E1 -9456.65,E2 -9456.65} C_VEL
LIN {X 0,Y 431.739,Z 989.079,A -85,B 0,C 180,E1 -9458.187,E2 -9458.187} C_VEL
LIN {X 0,Y 431.924,Z 982.168,A -85,B 0,C 180,E1 -9459.599,E2 -9459.599} C_VEL
LIN {X 0,Y 432.326,Z 973.644,A -85,B 0,C 180,E1 -9461.01,E2 -9461.01} C_VEL
LIN {X 0,Y 432.774,Z 964.93,A -85,B 0,C 180,E1 -9462.186,E2 -9462.186} C_VEL
LIN {X 0,Y 433.316,Z 955.319,A -85,B 0,C 180,E1 -9463.251,E2 -9463.251} C_VEL
LIN {X 0,Y 433.931,Z 943.634,A -85,B 0,C 180,E1 -9464.298,E2 -9464.298} C_VEL
LIN {X 0,Y 434.745,Z 932.109,A -85,B 0,C 180,E1 -9465.108,E2 -9465.108} C_VEL
LIN {X 0,Y 435.321,Z 920.269,A -85,B 0,C 180,E1 -9465.748,E2 -9465.748} C_VEL
LIN {X 0,Y 435.982,Z 906.71,A -85,B 0,C 180,E1 -9466.264,E2 -9466.264} C_VEL
LIN {X 0,Y 436.311,Z 893.285,A -85,B 0,C 180,E1 -9466.582,E2 -9466.582} C_VEL
LIN {X 0,Y 436.958,Z 819.379,A -85,B 0,C 180,E1 -9467.812,E2 -9467.812} C_VEL
LIN {X 0,Y 433.622,Z 788.488,A -85,B 0,C 180,E1 -9468.508,E2 -9468.508} C_VEL
LIN {X 0,Y 434.791,Z 763.257,A -85,B 0,C 180,E1 -9472.073,E2 -9472.073} C_VEL
LIN {X 0,Y 435.933,Z 741.786,A -85,B 0,C 180,E1 -9475.171,E2 -9475.171} C_VEL
LIN {X 0,Y 437.222,Z 722.173,A -85,B 0,C 180,E1 -9478.043,E2 -9478.043} C_VEL
LIN {X 0,Y 436.895,Z 718.671,A -85,B 0,C 180,E1 -9478.59,E2 -9478.59} C_VEL
LIN {X 0,Y 433.868,Z 705.149,A -85,B 0,C 180,E1 -9480.849,E2 -9480.849} C_VEL
LIN {X 0,Y 432.337,Z 698.731,A -85,B 0,C 180,E1 -9482.015,E2 -9482.015} C_VEL
LIN {X 0,Y 432.334,Z 698.627,A -85,B 0,C 180,E1 -9484.676,E2 -9484.676} C_VEL
LIN {X 0,Y 432.33,Z 698.631,A -85,B 0,C 180,E1 -9488.149,E2 -9488.149} C_VEL
LIN {X 0,Y 432.325,Z 698.631,A -85,B 0,C 180,E1 -9491.601,E2 -9491.601} C_VEL
LIN {X 0,Y 432.326,Z 698.632,A -85,B 0,C 180,E1 -9494.346,E2 -9494.346} C_VEL
LIN {X 0,Y 432.317,Z 698.633,A -85,B 0,C 180,E1 -9497.014,E2 -9497.014} C_VEL
LIN {X 0,Y 432.328,Z 698.622,A -85,B 0,C 180,E1 -9499.819,E2 -9499.819} C_VEL
LIN {X 0,Y 432.306,Z 698.634,A -85,B 0,C 180,E1 -9503.022,E2 -9503.022} C_VEL
LIN {X 0,Y 432.35,Z 698.625,A -85,B 0,C 180,E1 -9505.995,E2 -9505.995} C_VEL
LIN {X 0,Y 432.384,Z 698.625,A -85,B 0,C 180,E1 -9509.743,E2 -9509.743} C_VEL
LIN {X 0,Y 432.391,Z 698.628,A -85,B 0,C 180,E1 -9513.371,E2 -9513.371} C_VEL
LIN {X 0,Y 432.36,Z 698.627,A -85,B 0,C 180,E1 -9516.023,E2 -9516.023} C_VEL
LIN {X 0,Y 432.338,Z 698.625,A -85,B 0,C 180,E1 -9519.045,E2 -9519.045} C_VEL
LIN {X 0,Y 432.367,Z 698.623,A -85,B 0,C 180,E1 -9522.011,E2 -9522.011} C_VEL
LIN {X 0,Y 432.39,Z 698.621,A -85,B 0,C 180,E1 -9524.926,E2 -9524.926} C_VEL
LIN {X 0,Y 432.447,Z 698.615,A -85,B 0,C 180,E1 -9527.803,E2 -9527.803} C_VEL
LIN {X 0,Y 432.48,Z 698.606,A -85,B 0,C 180,E1 -9531.59,E2 -9531.59} C_VEL
LIN {X 0,Y 432.582,Z 698.598,A -85,B 0,C 180,E1 -9534.406,E2 -9534.406} C_VEL
LIN {X 0,Y 432.594,Z 698.601,A -85,B 0,C 180,E1 -9538.138,E2 -9538.138} C_VEL
LIN {X 0,Y 432.72,Z 698.58,A -85,B 0,C 180,E1 -9540,E2 -9540} C_VEL
LIN {X 0,Y 432.593,Z 698.598,A -85,B 0,C 180,E1 -9542.794,E2 -9542.794} C_VEL
LIN {X 0,Y 432.557,Z 698.606,A -85,B 0,C 180,E1 -9546.531,E2 -9546.531} C_VEL
LIN {X 0,Y 432.432,Z 698.616,A -85,B 0,C 180,E1 -9549.354,E2 -9549.354} C_VEL
LIN {X 0,Y 432.419,Z 698.619,A -85,B 0,C 180,E1 -9552.804,E2 -9552.804} C_VEL
LIN {X 0,Y 432.4,Z 698.618,A -85,B 0,C 180,E1 -9556.479,E2 -9556.479} C_VEL
LIN {X 0,Y 432.327,Z 698.628,A -85,B 0,C 180,E1 -9559.961,E2 -9559.961} C_VEL
LIN {X 0,Y 432.305,Z 698.627,A -85,B 0,C 180,E1 -9562.965,E2 -9562.965} C_VEL
LIN {X 0,Y 432.34,Z 698.63,A -85,B 0,C 180,E1 -9566.034,E2 -9566.034} C_VEL
LIN {X 0,Y 432.333,Z 698.625,A -85,B 0,C 180,E1 -9569.189,E2 -9569.189} C_VEL
LIN {X 0,Y 432.314,Z 698.626,A -85,B 0,C 180,E1 -9572.444,E2 -9572.444} C_VEL
LIN {X 0,Y 432.337,Z 698.628,A -85,B 0,C 180,E1 -9575.633,E2 -9575.633} C_VEL
LIN {X 0,Y 432.344,Z 698.624,A -85,B 0,C 180,E1 -9578.718,E2 -9578.718} C_VEL
LIN {X 0,Y 432.326,Z 698.634,A -85,B 0,C 180,E1 -9581.798,E2 -9581.798} C_VEL
LIN {X 0,Y 432.327,Z 698.632,A -85,B 0,C 180,E1 -9584.349,E2 -9584.349} C_VEL
LIN {X 0,Y 432.38,Z 698.812,A -85,B 0,C 180,E1 -9586.816,E2 -9586.816} C_VEL
LIN {X 0,Y 432.628,Z 699.89,A -85,B 0,C 180,E1 -9586.973,E2 -9586.973} C_VEL
LIN {X 0,Y 437.751,Z 712.971,A -85,B 0,C 180,E1 -9587.453,E2 -9587.453} C_VEL
LIN {X 0,Y 437.159,Z 780.221,A -85,B 0,C 180,E1 -9588.609,E2 -9588.609} C_VEL
LIN {X 0,Y 437.03,Z 793.572,A -85,B 0,C 180,E1 -9589.03,E2 -9589.03} C_VEL
LIN {X 0,Y 436.845,Z 805.835,A -85,B 0,C 180,E1 -9589.607,E2 -9589.607} C_VEL
LIN {X 0,Y 436.508,Z 817.558,A -85,B 0,C 180,E1 -9590.349,E2 -9590.349} C_VEL
LIN {X 0,Y 435.998,Z 828.05,A -85,B 0,C 180,E1 -9591.2,E2 -9591.2} C_VEL
LIN {X 0,Y 435.431,Z 838.582,A -85,B 0,C 180,E1 -9592.268,E2 -9592.268} C_VEL
LIN {X 0,Y 434.783,Z 848.218,A -85,B 0,C 180,E1 -9593.479,E2 -9593.479} C_VEL
LIN {X 0,Y 434.227,Z 855.783,A -85,B 0,C 180,E1 -9594.649,E2 -9594.649} C_VEL
LIN {X 0,Y 433.715,Z 863.501,A -85,B 0,C 180,E1 -9596.133,E2 -9596.133} C_VEL
LIN {X 0,Y 433.223,Z 869.693,A -85,B 0,C 180,E1 -9597.635,E2 -9597.635} C_VEL
LIN {X 0,Y 432.821,Z 875.127,A -85,B 0,C 180,E1 -9599.384,E2 -9599.384} C_VEL
LIN {X 0,Y 432.59,Z 878.376,A -85,B 0,C 180,E1 -9600.833,E2 -9600.833} C_VEL
LIN {X 0,Y 432.458,Z 880.093,A -85,B 0,C 180,E1 -9601.884,E2 -9601.884} C_VEL
LIN {X 0,Y 432.355,Z 881.644,A -85,B 0,C 180,E1 -9603.386,E2 -9603.386} C_VEL
LIN {X 0,Y 432.262,Z 882.198,A -85,B 0,C 180,E1 -9604.995,E2 -9604.995} C_VEL
LIN {X 0,Y 432.236,Z 881.925,A -85,B 0,C 180,E1 -9606.017,E2 -9606.017} C_VEL
LIN {X 0,Y 432.347,Z 880.223,A -85,B 0,C 180,E1 -9607.906,E2 -9607.906} C_VEL
LIN {X 0,Y 432.581,Z 877.371,A -85,B 0,C 180,E1 -9609.557,E2 -9609.557} C_VEL
LIN {X 0,Y 432.802,Z 873.623,A -85,B 0,C 180,E1 -9611.05,E2 -9611.05} C_VEL
LIN {X 0,Y 433.187,Z 868.653,A -85,B 0,C 180,E1 -9612.535,E2 -9612.535} C_VEL
LIN {X 0,Y 433.578,Z 862.385,A -85,B 0,C 180,E1 -9614.006,E2 -9614.006} C_VEL
LIN {X 0,Y 434.124,Z 854.536,A -85,B 0,C 180,E1 -9615.469,E2 -9615.469} C_VEL
LIN {X 0,Y 434.646,Z 846.064,A -85,B 0,C 180,E1 -9616.733,E2 -9616.733} C_VEL
LIN {X 0,Y 435.117,Z 838.04,A -85,B 0,C 180,E1 -9617.725,E2 -9617.725} C_VEL
LIN {X 0,Y 434.778,Z 833.629,A -85,B 0,C 180,E1 -9618.227,E2 -9618.227} C_VEL
LIN {X 0,Y 432.389,Z 826.328,A -85,B 0,C 180,E1 -9619.048,E2 -9619.048} C_VEL
LIN {X 0,Y 429.984,Z 818.506,A -85,B 0,C 180,E1 -9619.801,E2 -9619.801} C_VEL
LIN {X 0,Y 429.58,Z 813.31,A -85,B 0,C 180,E1 -9620.192,E2 -9620.192} C_VEL
LIN {X 0,Y 429.909,Z 801.28,A -85,B 0,C 180,E1 -9620.889,E2 -9620.889} C_VEL
LIN {X 0,Y 430.079,Z 788.264,A -85,B 0,C 180,E1 -9621.426,E2 -9621.426} C_VEL
LIN {X 0,Y 430.184,Z 775.776,A -85,B 0,C 180,E1 -9621.753,E2 -9621.753} C_VEL
LIN {X 0,Y 430.643,Z 713.831,A -85,B 0,C 180,E1 -9622.813,E2 -9622.813} C_VEL
LIN {X 0,Y 425.754,Z 700.736,A -85,B 0,C 180,E1 -9623.277,E2 -9623.277} C_VEL
LIN {X 0,Y 425.515,Z 699.628,A -85,B 0,C 180,E1 -9623.452,E2 -9623.452} C_VEL
LIN {X 0,Y 425.347,Z 699.496,A -85,B 0,C 180,E1 -9625.263,E2 -9625.263} C_VEL
LIN {X 0,Y 425.568,Z 699.475,A -85,B 0,C 180,E1 -9628.109,E2 -9628.109} C_VEL
LIN {X 0,Y 425.576,Z 699.473,A -85,B 0,C 180,E1 -9630.001,E2 -9630.001} C_VEL
LIN {X 0,Y 425.513,Z 699.482,A -85,B 0,C 180,E1 -9632.842,E2 -9632.842} C_VEL
LIN {X 0,Y 425.513,Z 699.48,A -85,B 0,C 180,E1 -9635.689,E2 -9635.689} C_VEL
LIN {X 0,Y 425.398,Z 699.498,A -85,B 0,C 180,E1 -9638.552,E2 -9638.552} C_VEL
LIN {X 0,Y 425.413,Z 699.494,A -85,B 0,C 180,E1 -9642.403,E2 -9642.403} C_VEL
LIN {X 0,Y 425.39,Z 699.492,A -85,B 0,C 180,E1 -9646.313,E2 -9646.313} C_VEL
LIN {X 0,Y 425.303,Z 699.495,A -85,B 0,C 180,E1 -9649.624,E2 -9649.624} C_VEL
LIN {X 0,Y 425.293,Z 699.505,A -85,B 0,C 180,E1 -9652.34,E2 -9652.34} C_VEL
LIN {X 0,Y 425.251,Z 699.503,A -85,B 0,C 180,E1 -9655.45,E2 -9655.45} C_VEL
LIN {X 0,Y 425.302,Z 699.503,A -85,B 0,C 180,E1 -9658.858,E2 -9658.858} C_VEL
LIN {X 0,Y 425.252,Z 699.507,A -85,B 0,C 180,E1 -9661.929,E2 -9661.929} C_VEL
LIN {X 0,Y 425.295,Z 699.491,A -85,B 0,C 180,E1 -9665.338,E2 -9665.338} C_VEL
LIN {X 0,Y 425.27,Z 699.508,A -85,B 0,C 180,E1 -9668.903,E2 -9668.903} C_VEL
LIN {X 0,Y 425.248,Z 699.513,A -85,B 0,C 180,E1 -9671.951,E2 -9671.951} C_VEL
LIN {X 0,Y 425.285,Z 699.509,A -85,B 0,C 180,E1 -9675.285,E2 -9675.285} C_VEL
LIN {X 0,Y 425.251,Z 699.51,A -85,B 0,C 180,E1 -9678.618,E2 -9678.618} C_VEL
LIN {X 0,Y 425.272,Z 699.511,A -85,B 0,C 180,E1 -9682.305,E2 -9682.305} C_VEL
LIN {X 0,Y 425.275,Z 699.513,A -85,B 0,C 180,E1 -9685.814,E2 -9685.814} C_VEL
LIN {X 0,Y 425.314,Z 699.638,A -85,B 0,C 180,E1 -9688.945,E2 -9688.945} C_VEL
LIN {X 0,Y 425.526,Z 700.644,A -85,B 0,C 180,E1 -9689.117,E2 -9689.117} C_VEL
LIN {X 0,Y 430.057,Z 713.765,A -85,B 0,C 180,E1 -9689.562,E2 -9689.562} C_VEL
LIN {X 0,Y 429.313,Z 775.624,A -85,B 0,C 180,E1 -9690.721,E2 -9690.721} C_VEL
LIN {X 0,Y 429.117,Z 787.092,A -85,B 0,C 180,E1 -9691.075,E2 -9691.075} C_VEL
LIN {X 0,Y 428.864,Z 798.063,A -85,B 0,C 180,E1 -9691.558,E2 -9691.558} C_VEL
LIN {X 0,Y 428.562,Z 808.498,A -85,B 0,C 180,E1 -9692.16,E2 -9692.16} C_VEL
LIN {X 0,Y 428.201,Z 817.164,A -85,B 0,C 180,E1 -9692.773,E2 -9692.773} C_VEL
LIN {X 0,Y 427.749,Z 827.373,A -85,B 0,C 180,E1 -9693.665,E2 -9693.665} C_VEL
LIN {X 0,Y 427.291,Z 835.805,A -85,B 0,C 180,E1 -9694.551,E2 -9694.551} C_VEL
LIN {X 0,Y 426.944,Z 843.137,A -85,B 0,C 180,E1 -9695.461,E2 -9695.461} C_VEL
LIN {X 0,Y 426.606,Z 849.966,A -85,B 0,C 180,E1 -9696.453,E2 -9696.453} C_VEL
LIN {X 0,Y 426.124,Z 857.16,A -85,B 0,C 180,E1 -9697.707,E2 -9697.707} C_VEL
LIN {X 0,Y 425.807,Z 863.088,A -85,B 0,C 180,E1 -9698.962,E2 -9698.962} C_VEL
LIN {X 0,Y 425.534,Z 868.206,A -85,B 0,C 180,E1 -9700.29,E2 -9700.29} C_VEL
LIN {X 0,Y 425.294,Z 872.498,A -85,B 0,C 180,E1 -9701.701,E2 -9701.701} C_VEL
LIN {X 0,Y 425.174,Z 874.947,A -85,B 0,C 180,E1 -9702.69,E2 -9702.69} C_VEL
LIN {X 0,Y 424.991,Z 878.174,A -85,B 0,C 180,E1 -9704.657,E2 -9704.657} C_VEL
LIN {X 0,Y 424.99,Z 879.233,A -85,B 0,C 180,E1 -9705.637,E2 -9705.637} C_VEL
LIN {X 0,Y 425.039,Z 879.869,A -85,B 0,C 180,E1 -9707.311,E2 -9707.311} C_VEL
LIN {X 0,Y 425.068,Z 879.564,A -85,B 0,C 180,E1 -9708.556,E2 -9708.556} C_VEL
LIN {X 0,Y 425.261,Z 877.561,A -85,B 0,C 180,E1 -9710.487,E2 -9710.487} C_VEL
LIN {X 0,Y 425.411,Z 876.04,A -85,B 0,C 180,E1 -9711.449,E2 -9711.449} C_VEL
LIN {X 0,Y 425.679,Z 872.773,A -85,B 0,C 180,E1 -9712.887,E2 -9712.887} C_VEL
LIN {X 0,Y 425.96,Z 868.402,A -85,B 0,C 180,E1 -9714.318,E2 -9714.318} C_VEL
LIN {X 0,Y 426.294,Z 862.781,A -85,B 0,C 180,E1 -9715.745,E2 -9715.745} C_VEL
LIN {X 0,Y 426.706,Z 857.041,A -85,B 0,C 180,E1 -9716.931,E2 -9716.931} C_VEL
LIN {X 0,Y 427.195,Z 850.096,A -85,B 0,C 180,E1 -9718.114,E2 -9718.114} C_VEL
LIN {X 0,Y 427.698,Z 841.668,A -85,B 0,C 180,E1 -9719.294,E2 -9719.294} C_VEL
LIN {X 0,Y 428.156,Z 833.598,A -85,B 0,C 180,E1 -9720.235,E2 -9720.235} C_VEL
LIN {X 0,Y 428.677,Z 825.011,A -85,B 0,C 180,E1 -9721.068,E2 -9721.068} C_VEL
LIN {X 0,Y 429.041,Z 816.38,A -85,B 0,C 180,E1 -9721.772,E2 -9721.772} C_VEL
LIN {X 0,Y 429.374,Z 805.823,A -85,B 0,C 180,E1 -9722.462,E2 -9722.462} C_VEL
LIN {X 0,Y 429.677,Z 795.424,A -85,B 0,C 180,E1 -9722.988,E2 -9722.988} C_VEL
LIN {X 0,Y 429.821,Z 784.494,A -85,B 0,C 180,E1 -9723.398,E2 -9723.398} C_VEL
LIN {X 0,Y 429.877,Z 771.575,A -85,B 0,C 180,E1 -9723.72,E2 -9723.72} C_VEL
LIN {X 0,Y 430.844,Z 713.938,A -85,B 0,C 180,E1 -9724.834,E2 -9724.834} C_VEL
LIN {X 0,Y 425.709,Z 700.47,A -85,B 0,C 180,E1 -9725.414,E2 -9725.414} C_VEL
LIN {X 0,Y 425.557,Z 699.575,A -85,B 0,C 180,E1 -9725.596,E2 -9725.596} C_VEL
LIN {X 0,Y 425.415,Z 699.494,A -85,B 0,C 180,E1 -9728.55,E2 -9728.55} C_VEL
LIN {X 0,Y 425.42,Z 699.495,A -85,B 0,C 180,E1 -9732.401,E2 -9732.401} C_VEL
LIN {X 0,Y 425.395,Z 699.498,A -85,B 0,C 180,E1 -9736.311,E2 -9736.311} C_VEL
LIN {X 0,Y 425.336,Z 699.502,A -85,B 0,C 180,E1 -9739.635,E2 -9739.635} C_VEL
LIN {X 0,Y 425.295,Z 699.509,A -85,B 0,C 180,E1 -9742.338,E2 -9742.338} C_VEL
LIN {X 0,Y 425.328,Z 699.506,A -85,B 0,C 180,E1 -9744.657,E2 -9744.657} C_VEL
LIN {X 0,Y 425.307,Z 699.505,A -85,B 0,C 180,E1 -9747.561,E2 -9747.561} C_VEL
LIN {X 0,Y 425.294,Z 699.509,A -85,B 0,C 180,E1 -9750.816,E2 -9750.816} C_VEL
LIN {X 0,Y 425.316,Z 699.504,A -85,B 0,C 180,E1 -9754.287,E2 -9754.287} C_VEL
LIN {X 0,Y 425.286,Z 699.508,A -85,B 0,C 180,E1 -9757.694,E2 -9757.694} C_VEL
LIN {X 0,Y 425.288,Z 699.508,A -85,B 0,C 180,E1 -9760.52,E2 -9760.52} C_VEL
LIN {X 0,Y 425.264,Z 699.513,A -85,B 0,C 180,E1 -9763.35,E2 -9763.35} C_VEL
LIN {X 0,Y 425.263,Z 699.511,A -85,B 0,C 180,E1 -9766.648,E2 -9766.648} C_VEL
LIN {X 0,Y 425.291,Z 699.509,A -85,B 0,C 180,E1 -9769.872,E2 -9769.872} C_VEL
LIN {X 0,Y 425.282,Z 699.507,A -85,B 0,C 180,E1 -9772.488,E2 -9772.488} C_VEL
LIN {X 0,Y 425.311,Z 699.507,A -85,B 0,C 180,E1 -9775.816,E2 -9775.816} C_VEL
LIN {X 0,Y 425.306,Z 699.669,A -85,B 0,C 180,E1 -9777.635,E2 -9777.635} C_VEL
LIN {X 0,Y 428.923,Z 714.893,A -85,B 0,C 180,E1 -9780.275,E2 -9780.275} C_VEL
LIN {X 0,Y 430.411,Z 722.119,A -85,B 0,C 180,E1 -9781.469,E2 -9781.469} C_VEL
LIN {X 0,Y 429.638,Z 735.869,A -85,B 0,C 180,E1 -9783.527,E2 -9783.527} C_VEL
LIN {X 0,Y 428.101,Z 761.564,A -85,B 0,C 180,E1 -9787.306,E2 -9787.306} C_VEL
LIN {X 0,Y 426.725,Z 788.622,A -85,B 0,C 180,E1 -9791.215,E2 -9791.215} C_VEL
LIN {X 0,Y 427.282,Z 794.076,A -85,B 0,C 180,E1 -9791.375,E2 -9791.375} C_VEL
LIN {X 0,Y 430.184,Z 822.063,A -85,B 0,C 180,E1 -9791.982,E2 -9791.982} C_VEL
LIN {X 0,Y 429.37,Z 899.952,A -85,B 0,C 180,E1 -9793.323,E2 -9793.323} C_VEL
LIN {X 0,Y 428.783,Z 913.812,A -85,B 0,C 180,E1 -9793.759,E2 -9793.759} C_VEL
LIN {X 0,Y 428.119,Z 926.29,A -85,B 0,C 180,E1 -9794.344,E2 -9794.344} C_VEL
LIN {X 0,Y 427.399,Z 938.268,A -85,B 0,C 180,E1 -9795.111,E2 -9795.111} C_VEL
LIN {X 0,Y 426.759,Z 948.766,A -85,B 0,C 180,E1 -9795.965,E2 -9795.965} C_VEL
LIN {X 0,Y 426.162,Z 959.181,A -85,B 0,C 180,E1 -9797.014,E2 -9797.014} C_VEL
LIN {X 0,Y 425.522,Z 967.909,A -85,B 0,C 180,E1 -9798.084,E2 -9798.084} C_VEL
LIN {X 0,Y 425.118,Z 975.998,A -85,B 0,C 180,E1 -9799.28,E2 -9799.28} C_VEL
LIN {X 0,Y 424.785,Z 983.93,A -85,B 0,C 180,E1 -9800.716,E2 -9800.716} C_VEL
LIN {X 0,Y 424.609,Z 991.238,A -85,B 0,C 180,E1 -9802.39,E2 -9802.39} C_VEL
LIN {X 0,Y 424.555,Z 995.562,A -85,B 0,C 180,E1 -9803.642,E2 -9803.642} C_VEL
LIN {X 0,Y 424.622,Z 999.854,A -85,B 0,C 180,E1 -9805.252,E2 -9805.252} C_VEL
LIN {X 0,Y 424.663,Z 1001.782,A -85,B 0,C 180,E1 -9806.203,E2 -9806.203} C_VEL
LIN {X 0,Y 424.616,Z 1003.215,A -85,B 0,C 180,E1 -9807.152,E2 -9807.152} C_VEL
LIN {X 0,Y 424.628,Z 1004.234,A -85,B 0,C 180,E1 -9808.102,E2 -9808.102} C_VEL
LIN {X 0,Y 424.638,Z 1004.848,A -85,B 0,C 180,E1 -9809.05,E2 -9809.05} C_VEL
LIN {X 0,Y 424.653,Z 1005.059,A -85,B 0,C 180,E1 -9809.999,E2 -9809.999} C_VEL
LIN {X 0,Y 424.642,Z 1004.817,A -85,B 0,C 180,E1 -9810.947,E2 -9810.947} C_VEL
LIN {X 0,Y 424.636,Z 1004.166,A -85,B 0,C 180,E1 -9811.895,E2 -9811.895} C_VEL
LIN {X 0,Y 424.623,Z 1003.11,A -85,B 0,C 180,E1 -9812.845,E2 -9812.845} C_VEL
LIN {X 0,Y 424.663,Z 1001.647,A -85,B 0,C 180,E1 -9813.794,E2 -9813.794} C_VEL
LIN {X 0,Y 424.597,Z 998.561,A -85,B 0,C 180,E1 -9815.222,E2 -9815.222} C_VEL
LIN {X 0,Y 424.558,Z 994.336,A -85,B 0,C 180,E1 -9816.674,E2 -9816.674} C_VEL
LIN {X 0,Y 424.697,Z 988.059,A -85,B 0,C 180,E1 -9818.324,E2 -9818.324} C_VEL
LIN {X 0,Y 424.874,Z 981.145,A -85,B 0,C 180,E1 -9819.76,E2 -9819.76} C_VEL
LIN {X 0,Y 425.275,Z 972.615,A -85,B 0,C 180,E1 -9821.195,E2 -9821.195} C_VEL
LIN {X 0,Y 425.814,Z 963.913,A -85,B 0,C 180,E1 -9822.388,E2 -9822.388} C_VEL
LIN {X 0,Y 426.396,Z 953.433,A -85,B 0,C 180,E1 -9823.558,E2 -9823.558} C_VEL
LIN {X 0,Y 426.98,Z 942.618,A -85,B 0,C 180,E1 -9824.536,E2 -9824.536} C_VEL
LIN {X 0,Y 427.85,Z 931.107,A -85,B 0,C 180,E1 -9825.358,E2 -9825.358} C_VEL
LIN {X 0,Y 428.457,Z 919.292,A -85,B 0,C 180,E1 -9826.007,E2 -9826.007} C_VEL
LIN {X 0,Y 429.123,Z 905.765,A -85,B 0,C 180,E1 -9826.531,E2 -9826.531} C_VEL
LIN {X 0,Y 429.495,Z 892.454,A -85,B 0,C 180,E1 -9826.853,E2 -9826.853} C_VEL
LIN {X 0,Y 430.124,Z 819.776,A -85,B 0,C 180,E1 -9828.085,E2 -9828.085} C_VEL
LIN {X 0,Y 426.657,Z 787.51,A -85,B 0,C 180,E1 -9828.822,E2 -9828.822} C_VEL
LIN {X 0,Y 427.908,Z 762.283,A -85,B 0,C 180,E1 -9832.447,E2 -9832.447} C_VEL
LIN {X 0,Y 429.186,Z 739.791,A -85,B 0,C 180,E1 -9835.758,E2 -9835.758} C_VEL
LIN {X 0,Y 430.339,Z 723.005,A -85,B 0,C 180,E1 -9838.267,E2 -9838.267} C_VEL
LIN {X 0,Y 429.111,Z 715.962,A -85,B 0,C 180,E1 -9839.427,E2 -9839.427} C_VEL
LIN {X 0,Y 425.81,Z 701.838,A -85,B 0,C 180,E1 -9841.879,E2 -9841.879} C_VEL
LIN {X 0,Y 425.288,Z 699.601,A -85,B 0,C 180,E1 -9842.336,E2 -9842.336} C_VEL
LIN {X 0,Y 425.293,Z 699.509,A -85,B 0,C 180,E1 -9845.334,E2 -9845.334} C_VEL
LIN {X 0,Y 425.287,Z 699.511,A -85,B 0,C 180,E1 -9849.041,E2 -9849.041} C_VEL
LIN {X 0,Y 425.267,Z 699.51,A -85,B 0,C 180,E1 -9852.652,E2 -9852.652} C_VEL
LIN {X 0,Y 425.261,Z 699.507,A -85,B 0,C 180,E1 -9856.044,E2 -9856.044} C_VEL
LIN {X 0,Y 425.268,Z 699.514,A -85,B 0,C 180,E1 -9858.621,E2 -9858.621} C_VEL
LIN {X 0,Y 425.304,Z 699.505,A -85,B 0,C 180,E1 -9861.102,E2 -9861.102} C_VEL
LIN {X 0,Y 425.291,Z 699.499,A -85,B 0,C 180,E1 -9864.663,E2 -9864.663} C_VEL
LIN {X 0,Y 425.256,Z 699.51,A -85,B 0,C 180,E1 -9868.072,E2 -9868.072} C_VEL
LIN {X 0,Y 425.327,Z 699.504,A -85,B 0,C 180,E1 -9871.368,E2 -9871.368} C_VEL
LIN {X 0,Y 425.284,Z 699.505,A -85,B 0,C 180,E1 -9874.554,E2 -9874.554} C_VEL
LIN {X 0,Y 425.276,Z 699.51,A -85,B 0,C 180,E1 -9877.661,E2 -9877.661} C_VEL
LIN {X 0,Y 425.35,Z 699.498,A -85,B 0,C 180,E1 -9880.704,E2 -9880.704} C_VEL
LIN {X 0,Y 425.387,Z 699.495,A -85,B 0,C 180,E1 -9883.688,E2 -9883.688} C_VEL
LIN {X 0,Y 425.4,Z 699.49,A -85,B 0,C 180,E1 -9887.598,E2 -9887.598} C_VEL
LIN {X 0,Y 425.43,Z 699.483,A -85,B 0,C 180,E1 -9891.45,E2 -9891.45} C_VEL
LIN {X 0,Y 425.538,Z 699.477,A -85,B 0,C 180,E1 -9894.313,E2 -9894.313} C_VEL
LIN {X 0,Y 425.564,Z 699.476,A -85,B 0,C 180,E1 -9898.107,E2 -9898.107} C_VEL
LIN {X 0,Y 425.69,Z 699.456,A -85,B 0,C 180,E1 -9900,E2 -9900} C_VEL
LIN {X 0,Y 425.544,Z 699.475,A -85,B 0,C 180,E1 -9902.84,E2 -9902.84} C_VEL
LIN {X 0,Y 425.516,Z 699.484,A -85,B 0,C 180,E1 -9906.639,E2 -9906.639} C_VEL
LIN {X 0,Y 425.39,Z 699.492,A -85,B 0,C 180,E1 -9909.51,E2 -9909.51} C_VEL
LIN {X 0,Y 425.381,Z 699.496,A -85,B 0,C 180,E1 -9912.904,E2 -9912.904} C_VEL
LIN {X 0,Y 425.349,Z 699.497,A -85,B 0,C 180,E1 -9916.605,E2 -9916.605} C_VEL
LIN {X 0,Y 425.317,Z 699.503,A -85,B 0,C 180,E1 -9919.636,E2 -9919.636} C_VEL
LIN {X 0,Y 425.276,Z 699.505,A -85,B 0,C 180,E1 -9922.34,E2 -9922.34} C_VEL
LIN {X 0,Y 425.309,Z 699.498,A -85,B 0,C 180,E1 -9924.658,E2 -9924.658} C_VEL
LIN {X 0,Y 425.335,Z 699.498,A -85,B 0,C 180,E1 -9927.559,E2 -9927.559} C_VEL
LIN {X 0,Y 425.278,Z 699.511,A -85,B 0,C 180,E1 -9930.817,E2 -9930.817} C_VEL
LIN {X 0,Y 425.303,Z 699.506,A -85,B 0,C 180,E1 -9934.289,E2 -9934.289} C_VEL
LIN {X 0,Y 425.278,Z 699.513,A -85,B 0,C 180,E1 -9937.695,E2 -9937.695} C_VEL
LIN {X 0,Y 425.276,Z 699.509,A -85,B 0,C 180,E1 -9940.522,E2 -9940.522} C_VEL
LIN {X 0,Y 425.25,Z 699.512,A -85,B 0,C 180,E1 -9943.352,E2 -9943.352} C_VEL
LIN {X 0,Y 425.304,Z 699.656,A -85,B 0,C 180,E1 -9946.473,E2 -9946.473} C_VEL
LIN {X 0,Y 425.504,Z 700.622,A -85,B 0,C 180,E1 -9946.638,E2 -9946.638} C_VEL
LIN {X 0,Y 431.052,Z 714.648,A -85,B 0,C 180,E1 -9947.174,E2 -9947.174} C_VEL
LIN {X 0,Y 430.418,Z 780.846,A -85,B 0,C 180,E1 -9948.327,E2 -9948.327} C_VEL
LIN {X 0,Y 430.304,Z 794.167,A -85,B 0,C 180,E1 -9948.748,E2 -9948.748} C_VEL
LIN {X 0,Y 430.104,Z 806.7,A -85,B 0,C 180,E1 -9949.343,E2 -9949.343} C_VEL
LIN {X 0,Y 429.752,Z 818.131,A -85,B 0,C 180,E1 -9950.071,E2 -9950.071} C_VEL
LIN {X 0,Y 429.235,Z 828.613,A -85,B 0,C 180,E1 -9950.925,E2 -9950.925} C_VEL
LIN {X 0,Y 428.633,Z 839.359,A -85,B 0,C 180,E1 -9952.025,E2 -9952.025} C_VEL
LIN {X 0,Y 427.975,Z 848.454,A -85,B 0,C 180,E1 -9953.173,E2 -9953.173} C_VEL
LIN {X 0,Y 427.315,Z 857.346,A -85,B 0,C 180,E1 -9954.569,E2 -9954.569} C_VEL
LIN {X 0,Y 426.791,Z 864.411,A -85,B 0,C 180,E1 -9955.954,E2 -9955.954} C_VEL
LIN {X 0,Y 426.381,Z 869.613,A -85,B 0,C 180,E1 -9957.207,E2 -9957.207} C_VEL
LIN {X 0,Y 425.974,Z 874.489,A -85,B 0,C 180,E1 -9958.68,E2 -9958.68} C_VEL
LIN {X 0,Y 425.678,Z 878.525,A -85,B 0,C 180,E1 -9960.312,E2 -9960.312} C_VEL
LIN {X 0,Y 425.506,Z 880.469,A -85,B 0,C 180,E1 -9961.383,E2 -9961.383} C_VEL
LIN {X 0,Y 425.33,Z 882.512,A -85,B 0,C 180,E1 -9963.162,E2 -9963.162} C_VEL
LIN {X 0,Y 425.257,Z 883.156,A -85,B 0,C 180,E1 -9964.554,E2 -9964.554} C_VEL
LIN {X 0,Y 425.23,Z 883.096,A -85,B 0,C 180,E1 -9965.596,E2 -9965.596} C_VEL
LIN {X 0,Y 425.234,Z 882.58,A -85,B 0,C 180,E1 -9966.632,E2 -9966.632} C_VEL
LIN {X 0,Y 425.314,Z 881.493,A -85,B 0,C 180,E1 -9967.724,E2 -9967.724} C_VEL
LIN {X 0,Y 425.429,Z 880.119,A -85,B 0,C 180,E1 -9968.69,E2 -9968.69} C_VEL
LIN {X 0,Y 425.673,Z 877.005,A -85,B 0,C 180,E1 -9970.237,E2 -9970.237} C_VEL
LIN {X 0,Y 425.981,Z 872.839,A -85,B 0,C 180,E1 -9971.733,E2 -9971.733} C_VEL
LIN {X 0,Y 426.39,Z 866.874,A -85,B 0,C 180,E1 -9973.355,E2 -9973.355} C_VEL
LIN {X 0,Y 426.918,Z 859.236,A -85,B 0,C 180,E1 -9974.974,E2 -9974.974} C_VEL
LIN {X 0,Y 427.561,Z 850.427,A -85,B 0,C 180,E1 -9976.431,E2 -9976.431} C_VEL
LIN {X 0,Y 428.139,Z 841.086,A -85,B 0,C 180,E1 -9977.68,E2 -9977.68} C_VEL
LIN {X 0,Y 428.732,Z 831.004,A -85,B 0,C 180,E1 -9978.769,E2 -9978.769} C_VEL
LIN {X 0,Y 429.309,Z 819.577,A -85,B 0,C 180,E1 -9979.747,E2 -9979.747} C_VEL
LIN {X 0,Y 429.58,Z 813.31,A -85,B 0,C 180,E1 -9980.192,E2 -9980.192} C_VEL
LIN {X 0,Y 429.168,Z 808.064,A -85,B 0,C 180,E1 -9980.553,E2 -9980.553} C_VEL
LIN {X 0,Y 426.616,Z 799.493,A -85,B 0,C 180,E1 -9981.132,E2 -9981.132} C_VEL
LIN {X 0,Y 423.964,Z 790.648,A -85,B 0,C 180,E1 -9981.615,E2 -9981.615} C_VEL
LIN {X 0,Y 423.382,Z 784.979,A -85,B 0,C 180,E1 -9981.817,E2 -9981.817} C_VEL
LIN {X 0,Y 423.403,Z 768.846,A -85,B 0,C 180,E1 -9982.161,E2 -9982.161} C_VEL
LIN {X 0,Y 423.911,Z 715.475,A -85,B 0,C 180,E1 -9983.083,E2 -9983.083} C_VEL
LIN {X 0,Y 418.706,Z 701.514,A -85,B 0,C 180,E1 -9983.587,E2 -9983.587} C_VEL
LIN {X 0,Y 418.465,Z 700.494,A -85,B 0,C 180,E1 -9983.765,E2 -9983.765} C_VEL
LIN {X 0,Y 418.536,Z 700.351,A -85,B 0,C 180,E1 -9988.077,E2 -9988.077} C_VEL
LIN {X 0,Y 418.411,Z 700.365,A -85,B 0,C 180,E1 -9990.964,E2 -9990.964} C_VEL
LIN {X 0,Y 418.47,Z 700.359,A -85,B 0,C 180,E1 -9992.889,E2 -9992.889} C_VEL
LIN {X 0,Y 418.474,Z 700.358,A -85,B 0,C 180,E1 -9995.785,E2 -9995.785} C_VEL
LIN {X 0,Y 418.371,Z 700.373,A -85,B 0,C 180,E1 -9998.697,E2 -9998.697} C_VEL
LIN {X 0,Y 418.359,Z 700.376,A -85,B 0,C 180,E1 -10002.616,E2 -10002.616} C_VEL
LIN {X 0,Y 418.296,Z 700.373,A -85,B 0,C 180,E1 -10005.596,E2 -10005.596} C_VEL
LIN {X 0,Y 418.254,Z 700.384,A -85,B 0,C 180,E1 -10008.62,E2 -10008.62} C_VEL
LIN {X 0,Y 418.235,Z 700.383,A -85,B 0,C 180,E1 -10011.698,E2 -10011.698} C_VEL
LIN {X 0,Y 418.251,Z 700.383,A -85,B 0,C 180,E1 -10014.853,E2 -10014.853} C_VEL
LIN {X 0,Y 418.205,Z 700.382,A -85,B 0,C 180,E1 -10018.071,E2 -10018.071} C_VEL
LIN {X 0,Y 418.239,Z 700.389,A -85,B 0,C 180,E1 -10021.019,E2 -10021.019} C_VEL
LIN {X 0,Y 418.233,Z 700.371,A -85,B 0,C 180,E1 -10023.68,E2 -10023.68} C_VEL
LIN {X 0,Y 418.237,Z 700.379,A -85,B 0,C 180,E1 -10027.226,E2 -10027.226} C_VEL
LIN {X 0,Y 418.212,Z 700.388,A -85,B 0,C 180,E1 -10030.951,E2 -10030.951} C_VEL
LIN {X 0,Y 418.187,Z 700.396,A -85,B 0,C 180,E1 -10033.726,E2 -10033.726} C_VEL
LIN {X 0,Y 418.204,Z 700.388,A -85,B 0,C 180,E1 -10036.447,E2 -10036.447} C_VEL
LIN {X 0,Y 418.212,Z 700.388,A -85,B 0,C 180,E1 -10039.134,E2 -10039.134} C_VEL
LIN {X 0,Y 418.233,Z 700.386,A -85,B 0,C 180,E1 -10042.775,E2 -10042.775} C_VEL
LIN {X 0,Y 418.226,Z 700.392,A -85,B 0,C 180,E1 -10046.32,E2 -10046.32} C_VEL
LIN {X 0,Y 418.262,Z 700.498,A -85,B 0,C 180,E1 -10048.664,E2 -10048.664} C_VEL
LIN {X 0,Y 418.455,Z 701.484,A -85,B 0,C 180,E1 -10048.845,E2 -10048.845} C_VEL
LIN {X 0,Y 423.28,Z 715.014,A -85,B 0,C 180,E1 -10049.323,E2 -10049.323} C_VEL
LIN {X 0,Y 422.41,Z 776.561,A -85,B 0,C 180,E1 -10050.503,E2 -10050.503} C_VEL
LIN {X 0,Y 422.225,Z 788.444,A -85,B 0,C 180,E1 -10050.882,E2 -10050.882} C_VEL
LIN {X 0,Y 422.002,Z 798.416,A -85,B 0,C 180,E1 -10051.325,E2 -10051.325} C_VEL
LIN {X 0,Y 421.712,Z 808.634,A -85,B 0,C 180,E1 -10051.914,E2 -10051.914} C_VEL
LIN {X 0,Y 421.305,Z 817.734,A -85,B 0,C 180,E1 -10052.559,E2 -10052.559} C_VEL
LIN {X 0,Y 420.845,Z 828.024,A -85,B 0,C 180,E1 -10053.466,E2 -10053.466} C_VEL
LIN {X 0,Y 420.422,Z 835.451,A -85,B 0,C 180,E1 -10054.238,E2 -10054.238} C_VEL
LIN {X 0,Y 420.008,Z 843.758,A -85,B 0,C 180,E1 -10055.271,E2 -10055.271} C_VEL
LIN {X 0,Y 419.664,Z 850.784,A -85,B 0,C 180,E1 -10056.301,E2 -10056.301} C_VEL
LIN {X 0,Y 419.155,Z 858.021,A -85,B 0,C 180,E1 -10057.576,E2 -10057.576} C_VEL
LIN {X 0,Y 418.831,Z 863.988,A -85,B 0,C 180,E1 -10058.852,E2 -10058.852} C_VEL
LIN {X 0,Y 418.556,Z 868.831,A -85,B 0,C 180,E1 -10060.105,E2 -10060.105} C_VEL
LIN {X 0,Y 418.337,Z 872.847,A -85,B 0,C 180,E1 -10061.385,E2 -10061.385} C_VEL
LIN {X 0,Y 418.181,Z 875.319,A -85,B 0,C 180,E1 -10062.391,E2 -10062.391} C_VEL
LIN {X 0,Y 417.992,Z 878.921,A -85,B 0,C 180,E1 -10064.394,E2 -10064.394} C_VEL
LIN {X 0,Y 417.98,Z 880.019,A -85,B 0,C 180,E1 -10065.391,E2 -10065.391} C_VEL
LIN {X 0,Y 417.977,Z 880.722,A -85,B 0,C 180,E1 -10066.385,E2 -10066.385} C_VEL
LIN {X 0,Y 418.043,Z 880.918,A -85,B 0,C 180,E1 -10067.376,E2 -10067.376} C_VEL
LIN {X 0,Y 418.039,Z 880.726,A -85,B 0,C 180,E1 -10068.361,E2 -10068.361} C_VEL
LIN {X 0,Y 418.235,Z 879.011,A -85,B 0,C 180,E1 -10070.326,E2 -10070.326} C_VEL
LIN {X 0,Y 418.402,Z 877.518,A -85,B 0,C 180,E1 -10071.305,E2 -10071.305} C_VEL
LIN {X 0,Y 418.674,Z 874.437,A -85,B 0,C 180,E1 -10072.767,E2 -10072.767} C_VEL
LIN {X 0,Y 418.971,Z 870.286,A -85,B 0,C 180,E1 -10074.223,E2 -10074.223} C_VEL
LIN {X 0,Y 419.395,Z 863.845,A -85,B 0,C 180,E1 -10075.916,E2 -10075.916} C_VEL
LIN {X 0,Y 419.828,Z 858.115,A -85,B 0,C 180,E1 -10077.121,E2 -10077.121} C_VEL
LIN {X 0,Y 420.355,Z 851.179,A -85,B 0,C 180,E1 -10078.323,E2 -10078.323} C_VEL
LIN {X 0,Y 420.892,Z 842.77,A -85,B 0,C 180,E1 -10079.521,E2 -10079.521} C_VEL
LIN {X 0,Y 421.39,Z 834.687,A -85,B 0,C 180,E1 -10080.478,E2 -10080.478} C_VEL
LIN {X 0,Y 421.943,Z 826.078,A -85,B 0,C 180,E1 -10081.324,E2 -10081.324} C_VEL
LIN {X 0,Y 422.312,Z 817.593,A -85,B 0,C 180,E1 -10082.026,E2 -10082.026} C_VEL
LIN {X 0,Y 422.632,Z 807.893,A -85,B 0,C 180,E1 -10082.681,E2 -10082.681} C_VEL
LIN {X 0,Y 422.966,Z 796.926,A -85,B 0,C 180,E1 -10083.252,E2 -10083.252} C_VEL
LIN {X 0,Y 423.124,Z 786.535,A -85,B 0,C 180,E1 -10083.657,E2 -10083.657} C_VEL
LIN {X 0,Y 423.157,Z 773.984,A -85,B 0,C 180,E1 -10083.988,E2 -10083.988} C_VEL
LIN {X 0,Y 424.101,Z 715.003,A -85,B 0,C 180,E1 -10085.17,E2 -10085.17} C_VEL
LIN {X 0,Y 418.711,Z 701.36,A -85,B 0,C 180,E1 -10085.795,E2 -10085.795} C_VEL
LIN {X 0,Y 418.511,Z 700.442,A -85,B 0,C 180,E1 -10085.994,E2 -10085.994} C_VEL
LIN {X 0,Y 418.385,Z 700.37,A -85,B 0,C 180,E1 -10088.695,E2 -10088.695} C_VEL
LIN {X 0,Y 418.322,Z 700.376,A -85,B 0,C 180,E1 -10091.631,E2 -10091.631} C_VEL
LIN {X 0,Y 418.31,Z 700.381,A -85,B 0,C 180,E1 -10094.597,E2 -10094.597} C_VEL
LIN {X 0,Y 418.287,Z 700.38,A -85,B 0,C 180,E1 -10097.604,E2 -10097.604} C_VEL
LIN {X 0,Y 418.257,Z 700.387,A -85,B 0,C 180,E1 -10100.663,E2 -10100.663} C_VEL
LIN {X 0,Y 418.282,Z 700.379,A -85,B 0,C 180,E1 -10103.781,E2 -10103.781} C_VEL
LIN {X 0,Y 418.273,Z 700.384,A -85,B 0,C 180,E1 -10107.058,E2 -10107.058} C_VEL
LIN {X 0,Y 418.249,Z 700.386,A -85,B 0,C 180,E1 -10110.272,E2 -10110.272} C_VEL
LIN {X 0,Y 418.254,Z 700.384,A -85,B 0,C 180,E1 -10113.677,E2 -10113.677} C_VEL
LIN {X 0,Y 418.247,Z 700.388,A -85,B 0,C 180,E1 -10117.223,E2 -10117.223} C_VEL
LIN {X 0,Y 418.258,Z 700.385,A -85,B 0,C 180,E1 -10119.681,E2 -10119.681} C_VEL
LIN {X 0,Y 418.236,Z 700.386,A -85,B 0,C 180,E1 -10122.32,E2 -10122.32} C_VEL
LIN {X 0,Y 418.242,Z 700.387,A -85,B 0,C 180,E1 -10125.108,E2 -10125.108} C_VEL
LIN {X 0,Y 418.246,Z 700.388,A -85,B 0,C 180,E1 -10127.766,E2 -10127.766} C_VEL
LIN {X 0,Y 418.248,Z 700.383,A -85,B 0,C 180,E1 -10130.62,E2 -10130.62} C_VEL
LIN {X 0,Y 418.247,Z 700.386,A -85,B 0,C 180,E1 -10133.975,E2 -10133.975} C_VEL
LIN {X 0,Y 418.276,Z 700.549,A -85,B 0,C 180,E1 -10137.333,E2 -10137.333} C_VEL
LIN {X 0,Y 422.147,Z 716.935,A -85,B 0,C 180,E1 -10140.223,E2 -10140.223} C_VEL
LIN {X 0,Y 423.542,Z 724.421,A -85,B 0,C 180,E1 -10141.477,E2 -10141.477} C_VEL
LIN {X 0,Y 422.254,Z 743.483,A -85,B 0,C 180,E1 -10144.357,E2 -10144.357} C_VEL
LIN {X 0,Y 420.972,Z 763.98,A -85,B 0,C 180,E1 -10147.418,E2 -10147.418} C_VEL
LIN {X 0,Y 419.746,Z 787.73,A -85,B 0,C 180,E1 -10150.911,E2 -10150.911} C_VEL
LIN {X 0,Y 421.69,Z 806.221,A -85,B 0,C 180,E1 -10151.356,E2 -10151.356} C_VEL
LIN {X 0,Y 423.393,Z 822.939,A -85,B 0,C 180,E1 -10151.723,E2 -10151.723} C_VEL
LIN {X 0,Y 422.566,Z 898.664,A -85,B 0,C 180,E1 -10153.046,E2 -10153.046} C_VEL
LIN {X 0,Y 422,Z 911.858,A -85,B 0,C 180,E1 -10153.459,E2 -10153.459} C_VEL
LIN {X 0,Y 421.21,Z 925.146,A -85,B 0,C 180,E1 -10154.08,E2 -10154.08} C_VEL
LIN {X 0,Y 420.471,Z 937.162,A -85,B 0,C 180,E1 -10154.859,E2 -10154.859} C_VEL
LIN {X 0,Y 419.835,Z 947.419,A -85,B 0,C 180,E1 -10155.704,E2 -10155.704} C_VEL
LIN {X 0,Y 419.162,Z 958.221,A -85,B 0,C 180,E1 -10156.806,E2 -10156.806} C_VEL
LIN {X 0,Y 418.519,Z 966.846,A -85,B 0,C 180,E1 -10157.882,E2 -10157.882} C_VEL
LIN {X 0,Y 418.092,Z 974.945,A -85,B 0,C 180,E1 -10159.098,E2 -10159.098} C_VEL
LIN {X 0,Y 417.736,Z 982.889,A -85,B 0,C 180,E1 -10160.557,E2 -10160.557} C_VEL
LIN {X 0,Y 417.571,Z 988.323,A -85,B 0,C 180,E1 -10161.774,E2 -10161.774} C_VEL
LIN {X 0,Y 417.486,Z 993.891,A -85,B 0,C 180,E1 -10163.322,E2 -10163.322} C_VEL
LIN {X 0,Y 417.578,Z 998.837,A -85,B 0,C 180,E1 -10165.171,E2 -10165.171} C_VEL
LIN {X 0,Y 417.627,Z 1000.767,A -85,B 0,C 180,E1 -10166.139,E2 -10166.139} C_VEL
LIN {X 0,Y 417.576,Z 1002.203,A -85,B 0,C 180,E1 -10167.104,E2 -10167.104} C_VEL
LIN {X 0,Y 417.591,Z 1003.224,A -85,B 0,C 180,E1 -10168.07,E2 -10168.07} C_VEL
LIN {X 0,Y 417.606,Z 1003.841,A -85,B 0,C 180,E1 -10169.034,E2 -10169.034} C_VEL
LIN {X 0,Y 417.625,Z 1004.052,A -85,B 0,C 180,E1 -10169.999,E2 -10169.999} C_VEL
LIN {X 0,Y 417.611,Z 1003.811,A -85,B 0,C 180,E1 -10170.963,E2 -10170.963} C_VEL
LIN {X 0,Y 417.599,Z 1003.158,A -85,B 0,C 180,E1 -10171.927,E2 -10171.927} C_VEL
LIN {X 0,Y 417.582,Z 1002.101,A -85,B 0,C 180,E1 -10172.893,E2 -10172.893} C_VEL
LIN {X 0,Y 417.628,Z 1000.637,A -85,B 0,C 180,E1 -10173.858,E2 -10173.858} C_VEL
LIN {X 0,Y 417.539,Z 997.546,A -85,B 0,C 180,E1 -10175.31,E2 -10175.31} C_VEL
LIN {X 0,Y 417.497,Z 993.386,A -85,B 0,C 180,E1 -10176.766,E2 -10176.766} C_VEL
LIN {X 0,Y 417.631,Z 987.037,A -85,B 0,C 180,E1 -10178.466,E2 -10178.466} C_VEL
LIN {X 0,Y 417.823,Z 980.12,A -85,B 0,C 180,E1 -10179.926,E2 -10179.926} C_VEL
LIN {X 0,Y 418.249,Z 971.589,A -85,B 0,C 180,E1 -10181.386,E2 -10181.386} C_VEL
LIN {X 0,Y 418.858,Z 962.896,A -85,B 0,C 180,E1 -10182.597,E2 -10182.597} C_VEL
LIN {X 0,Y 419.389,Z 953.372,A -85,B 0,C 180,E1 -10183.69,E2 -10183.69} C_VEL
LIN {X 0,Y 419.956,Z 943.053,A -85,B 0,C 180,E1 -10184.661,E2 -10184.661} C_VEL
LIN {X 0,Y 420.851,Z 931.894,A -85,B 0,C 180,E1 -10185.496,E2 -10185.496} C_VEL
LIN {X 0,Y 421.538,Z 919.557,A -85,B 0,C 180,E1 -10186.214,E2 -10186.214} C_VEL
LIN {X 0,Y 422.252,Z 906.707,A -85,B 0,C 180,E1 -10186.746,E2 -10186.746} C_VEL
LIN {X 0,Y 422.668,Z 893.211,A -85,B 0,C 180,E1 -10187.102,E2 -10187.102} C_VEL
LIN {X 0,Y 423.403,Z 820.813,A -85,B 0,C 180,E1 -10188.354,E2 -10188.354} C_VEL
LIN {X 0,Y 419.717,Z 786.34,A -85,B 0,C 180,E1 -10189.162,E2 -10189.162} C_VEL
LIN {X 0,Y 420.916,Z 763.014,A -85,B 0,C 180,E1 -10192.582,E2 -10192.582} C_VEL
LIN {X 0,Y 422.248,Z 741.014,A -85,B 0,C 180,E1 -10195.881,E2 -10195.881} C_VEL
LIN {X 0,Y 423.404,Z 723.762,A -85,B 0,C 180,E1 -10198.512,E2 -10198.512} C_VEL
LIN {X 0,Y 420.884,Z 711.512,A -85,B 0,C 180,E1 -10200.615,E2 -10200.615} C_VEL
LIN {X 0,Y 418.251,Z 700.506,A -85,B 0,C 180,E1 -10202.638,E2 -10202.638} C_VEL
LIN {X 0,Y 418.253,Z 700.382,A -85,B 0,C 180,E1 -10204.84,E2 -10204.84} C_VEL
LIN {X 0,Y 418.247,Z 700.386,A -85,B 0,C 180,E1 -10208.44,E2 -10208.44} C_VEL
LIN {X 0,Y 418.214,Z 700.391,A -85,B 0,C 180,E1 -10210.947,E2 -10210.947} C_VEL
LIN {X 0,Y 418.202,Z 700.388,A -85,B 0,C 180,E1 -10213.728,E2 -10213.728} C_VEL
LIN {X 0,Y 418.208,Z 700.385,A -85,B 0,C 180,E1 -10216.448,E2 -10216.448} C_VEL
LIN {X 0,Y 418.215,Z 700.385,A -85,B 0,C 180,E1 -10219.129,E2 -10219.129} C_VEL
LIN {X 0,Y 418.225,Z 700.386,A -85,B 0,C 180,E1 -10222.164,E2 -10222.164} C_VEL
LIN {X 0,Y 418.256,Z 700.379,A -85,B 0,C 180,E1 -10225.419,E2 -10225.419} C_VEL
LIN {X 0,Y 418.206,Z 700.389,A -85,B 0,C 180,E1 -10228.603,E2 -10228.603} C_VEL
LIN {X 0,Y 418.285,Z 700.378,A -85,B 0,C 180,E1 -10231.936,E2 -10231.936} C_VEL
LIN {X 0,Y 418.278,Z 700.38,A -85,B 0,C 180,E1 -10235.162,E2 -10235.162} C_VEL
LIN {X 0,Y 418.222,Z 700.382,A -85,B 0,C 180,E1 -10238.303,E2 -10238.303} C_VEL
LIN {X 0,Y 418.272,Z 700.384,A -85,B 0,C 180,E1 -10241.383,E2 -10241.383} C_VEL
LIN {X 0,Y 418.299,Z 700.378,A -85,B 0,C 180,E1 -10244.406,E2 -10244.406} C_VEL
LIN {X 0,Y 418.343,Z 700.367,A -85,B 0,C 180,E1 -10247.385,E2 -10247.385} C_VEL
LIN {X 0,Y 418.329,Z 700.37,A -85,B 0,C 180,E1 -10250.328,E2 -10250.328} C_VEL
LIN {X 0,Y 418.475,Z 700.354,A -85,B 0,C 180,E1 -10253.249,E2 -10253.249} C_VEL
LIN {X 0,Y 418.329,Z 700.368,A -85,B 0,C 180,E1 -10255.182,E2 -10255.182} C_VEL
LIN {X 0,Y 418.533,Z 700.351,A -85,B 0,C 180,E1 -10258.076,E2 -10258.076} C_VEL
LIN {X 0,Y 418.66,Z 700.331,A -85,B 0,C 180,E1 -10260,E2 -10260} C_VEL
LIN {X 0,Y 418.498,Z 700.352,A -85,B 0,C 180,E1 -10262.888,E2 -10262.888} C_VEL
LIN {X 0,Y 418.479,Z 700.359,A -85,B 0,C 180,E1 -10266.751,E2 -10266.751} C_VEL
LIN {X 0,Y 418.388,Z 700.366,A -85,B 0,C 180,E1 -10268.696,E2 -10268.696} C_VEL
LIN {X 0,Y 418.305,Z 700.374,A -85,B 0,C 180,E1 -10271.632,E2 -10271.632} C_VEL
LIN {X 0,Y 418.291,Z 700.382,A -85,B 0,C 180,E1 -10274.598,E2 -10274.598} C_VEL
LIN {X 0,Y 418.274,Z 700.381,A -85,B 0,C 180,E1 -10277.605,E2 -10277.605} C_VEL
LIN {X 0,Y 418.238,Z 700.386,A -85,B 0,C 180,E1 -10280.664,E2 -10280.664} C_VEL
LIN {X 0,Y 418.262,Z 700.372,A -85,B 0,C 180,E1 -10283.783,E2 -10283.783} C_VEL
LIN {X 0,Y 418.3,Z 700.382,A -85,B 0,C 180,E1 -10287.072,E2 -10287.072} C_VEL
LIN {X 0,Y 418.235,Z 700.388,A -85,B 0,C 180,E1 -10290.273,E2 -10290.273} C_VEL
LIN {X 0,Y 418.24,Z 700.386,A -85,B 0,C 180,E1 -10293.678,E2 -10293.678} C_VEL
LIN {X 0,Y 418.237,Z 700.387,A -85,B 0,C 180,E1 -10297.225,E2 -10297.225} C_VEL
LIN {X 0,Y 418.248,Z 700.387,A -85,B 0,C 180,E1 -10299.683,E2 -10299.683} C_VEL
LIN {X 0,Y 418.222,Z 700.39,A -85,B 0,C 180,E1 -10302.323,E2 -10302.323} C_VEL
LIN {X 0,Y 418.249,Z 700.487,A -85,B 0,C 180,E1 -10306.109,E2 -10306.109} C_VEL
LIN {X 0,Y 418.456,Z 701.36,A -85,B 0,C 180,E1 -10306.292,E2 -10306.292} C_VEL
LIN {X 0,Y 424.31,Z 716.159,A -85,B 0,C 180,E1 -10306.88,E2 -10306.88} C_VEL
LIN {X 0,Y 423.687,Z 781.22,A -85,B 0,C 180,E1 -10308.032,E2 -10308.032} C_VEL
LIN {X 0,Y 423.584,Z 794.307,A -85,B 0,C 180,E1 -10308.438,E2 -10308.438} C_VEL
LIN {X 0,Y 423.383,Z 806.862,A -85,B 0,C 180,E1 -10309.031,E2 -10309.031} C_VEL
LIN {X 0,Y 423.04,Z 817.988,A -85,B 0,C 180,E1 -10309.735,E2 -10309.735} C_VEL
LIN {X 0,Y 422.473,Z 829.185,A -85,B 0,C 180,E1 -10310.641,E2 -10310.641} C_VEL
LIN {X 0,Y 421.886,Z 838.966,A -85,B 0,C 180,E1 -10311.638,E2 -10311.638} C_VEL
LIN {X 0,Y 421.135,Z 849.183,A -85,B 0,C 180,E1 -10312.927,E2 -10312.927} C_VEL
LIN {X 0,Y 420.522,Z 857.344,A -85,B 0,C 180,E1 -10314.203,E2 -10314.203} C_VEL
LIN {X 0,Y 419.959,Z 864.62,A -85,B 0,C 180,E1 -10315.613,E2 -10315.613} C_VEL
LIN {X 0,Y 419.373,Z 871.224,A -85,B 0,C 180,E1 -10317.229,E2 -10317.229} C_VEL
LIN {X 0,Y 418.944,Z 876.237,A -85,B 0,C 180,E1 -10318.821,E2 -10318.821} C_VEL
LIN {X 0,Y 418.667,Z 879.746,A -85,B 0,C 180,E1 -10320.319,E2 -10320.319} C_VEL
LIN {X 0,Y 418.431,Z 882.382,A -85,B 0,C 180,E1 -10321.949,E2 -10321.949} C_VEL
LIN {X 0,Y 418.338,Z 883.453,A -85,B 0,C 180,E1 -10323.027,E2 -10323.027} C_VEL
LIN {X 0,Y 418.261,Z 884.068,A -85,B 0,C 180,E1 -10324.097,E2 -10324.097} C_VEL
LIN {X 0,Y 418.208,Z 884.198,A -85,B 0,C 180,E1 -10325.159,E2 -10325.159} C_VEL
LIN {X 0,Y 418.202,Z 883.844,A -85,B 0,C 180,E1 -10326.215,E2 -10326.215} C_VEL
LIN {X 0,Y 418.267,Z 882.757,A -85,B 0,C 180,E1 -10327.541,E2 -10327.541} C_VEL
LIN {X 0,Y 418.511,Z 880.03,A -85,B 0,C 180,E1 -10329.352,E2 -10329.352} C_VEL
LIN {X 0,Y 418.775,Z 876.523,A -85,B 0,C 180,E1 -10330.899,E2 -10330.899} C_VEL
LIN {X 0,Y 419.148,Z 871.847,A -85,B 0,C 180,E1 -10332.435,E2 -10332.435} C_VEL
LIN {X 0,Y 419.596,Z 865.859,A -85,B 0,C 180,E1 -10333.958,E2 -10333.958} C_VEL
LIN {X 0,Y 420.133,Z 858.345,A -85,B 0,C 180,E1 -10335.47,E2 -10335.47} C_VEL
LIN {X 0,Y 420.716,Z 850.653,A -85,B 0,C 180,E1 -10336.723,E2 -10336.723} C_VEL
LIN {X 0,Y 421.312,Z 841.358,A -85,B 0,C 180,E1 -10337.966,E2 -10337.966} C_VEL
LIN {X 0,Y 421.964,Z 830.315,A -85,B 0,C 180,E1 -10339.142,E2 -10339.142} C_VEL
LIN {X 0,Y 422.549,Z 819.409,A -85,B 0,C 180,E1 -10340.065,E2 -10340.065} C_VEL
LIN {X 0,Y 422.995,Z 807.42,A -85,B 0,C 180,E1 -10340.86,E2 -10340.86} C_VEL
LIN {X 0,Y 423.253,Z 794.242,A -85,B 0,C 180,E1 -10341.497,E2 -10341.497} C_VEL
LIN {X 0,Y 423.382,Z 784.979,A -85,B 0,C 180,E1 -10341.817,E2 -10341.817} C_VEL
LIN {X 0,Y 422.834,Z 779.236,A -85,B 0,C 180,E1 -10341.989,E2 -10341.989} C_VEL
LIN {X 0,Y 417.384,Z 760.66,A -85,B 0,C 180,E1 -10342.57,E2 -10342.57} C_VEL
LIN {X 0,Y 416.764,Z 754.865,A -85,B 0,C 180,E1 -10342.698,E2 -10342.698} C_VEL
LIN {X 0,Y 417.113,Z 716.813,A -85,B 0,C 180,E1 -10343.369,E2 -10343.369} C_VEL
LIN {X 0,Y 411.574,Z 702.043,A -85,B 0,C 180,E1 -10343.932,E2 -10343.932} C_VEL
LIN {X 0,Y 411.469,Z 701.299,A -85,B 0,C 180,E1 -10344.119,E2 -10344.119} C_VEL
LIN {X 0,Y 411.505,Z 701.227,A -85,B 0,C 180,E1 -10348.044,E2 -10348.044} C_VEL
LIN {X 0,Y 411.381,Z 701.241,A -85,B 0,C 180,E1 -10350.98,E2 -10350.98} C_VEL
LIN {X 0,Y 411.428,Z 701.236,A -85,B 0,C 180,E1 -10352.939,E2 -10352.939} C_VEL
LIN {X 0,Y 411.395,Z 701.236,A -85,B 0,C 180,E1 -10356.869,E2 -10356.869} C_VEL
LIN {X 0,Y 411.277,Z 701.252,A -85,B 0,C 180,E1 -10359.841,E2 -10359.841} C_VEL
LIN {X 0,Y 411.31,Z 701.248,A -85,B 0,C 180,E1 -10363.104,E2 -10363.104} C_VEL
LIN {X 0,Y 411.263,Z 701.259,A -85,B 0,C 180,E1 -10366.89,E2 -10366.89} C_VEL
LIN {X 0,Y 411.21,Z 701.25,A -85,B 0,C 180,E1 -10369.989,E2 -10369.989} C_VEL
LIN {X 0,Y 411.193,Z 701.266,A -85,B 0,C 180,E1 -10373.15,E2 -10373.15} C_VEL
LIN {X 0,Y 411.164,Z 701.255,A -85,B 0,C 180,E1 -10376.387,E2 -10376.387} C_VEL
LIN {X 0,Y 411.198,Z 701.262,A -85,B 0,C 180,E1 -10379.714,E2 -10379.714} C_VEL
LIN {X 0,Y 411.209,Z 701.253,A -85,B 0,C 180,E1 -10383.157,E2 -10383.157} C_VEL
LIN {X 0,Y 411.193,Z 701.25,A -85,B 0,C 180,E1 -10386.552,E2 -10386.552} C_VEL
LIN {X 0,Y 411.169,Z 701.269,A -85,B 0,C 180,E1 -10389.72,E2 -10389.72} C_VEL
LIN {X 0,Y 411.125,Z 701.272,A -85,B 0,C 180,E1 -10393.141,E2 -10393.141} C_VEL
LIN {X 0,Y 411.167,Z 701.27,A -85,B 0,C 180,E1 -10395.883,E2 -10395.883} C_VEL
LIN {X 0,Y 411.152,Z 701.267,A -85,B 0,C 180,E1 -10398.775,E2 -10398.775} C_VEL
LIN {X 0,Y 411.182,Z 701.268,A -85,B 0,C 180,E1 -10402.024,E2 -10402.024} C_VEL
LIN {X 0,Y 411.194,Z 701.263,A -85,B 0,C 180,E1 -10405.127,E2 -10405.127} C_VEL
LIN {X 0,Y 411.215,Z 701.392,A -85,B 0,C 180,E1 -10408.401,E2 -10408.401} C_VEL
LIN {X 0,Y 411.419,Z 702.352,A -85,B 0,C 180,E1 -10408.576,E2 -10408.576} C_VEL
LIN {X 0,Y 416.413,Z 716.274,A -85,B 0,C 180,E1 -10409.077,E2 -10409.077} C_VEL
LIN {X 0,Y 415.535,Z 777.528,A -85,B 0,C 180,E1 -10410.279,E2 -10410.279} C_VEL
LIN {X 0,Y 415.362,Z 788.997,A -85,B 0,C 180,E1 -10410.649,E2 -10410.649} C_VEL
LIN {X 0,Y 415.068,Z 799.943,A -85,B 0,C 180,E1 -10411.146,E2 -10411.146} C_VEL
LIN {X 0,Y 414.836,Z 809.099,A -85,B 0,C 180,E1 -10411.682,E2 -10411.682} C_VEL
LIN {X 0,Y 414.349,Z 819.944,A -85,B 0,C 180,E1 -10412.478,E2 -10412.478} C_VEL
LIN {X 0,Y 413.942,Z 828.674,A -85,B 0,C 180,E1 -10413.261,E2 -10413.261} C_VEL
LIN {X 0,Y 413.452,Z 836.943,A -85,B 0,C 180,E1 -10414.141,E2 -10414.141} C_VEL
LIN {X 0,Y 413.089,Z 844.529,A -85,B 0,C 180,E1 -10415.097,E2 -10415.097} C_VEL
LIN {X 0,Y 412.573,Z 853.087,A -85,B 0,C 180,E1 -10416.402,E2 -10416.402} C_VEL
LIN {X 0,Y 412.191,Z 858.925,A -85,B 0,C 180,E1 -10417.45,E2 -10417.45} C_VEL
LIN {X 0,Y 411.835,Z 864.888,A -85,B 0,C 180,E1 -10418.738,E2 -10418.738} C_VEL
LIN {X 0,Y 411.552,Z 869.818,A -85,B 0,C 180,E1 -10420.029,E2 -10420.029} C_VEL
LIN {X 0,Y 411.289,Z 874.43,A -85,B 0,C 180,E1 -10421.571,E2 -10421.571} C_VEL
LIN {X 0,Y 411.103,Z 877.857,A -85,B 0,C 180,E1 -10423.105,E2 -10423.105} C_VEL
LIN {X 0,Y 410.992,Z 879.632,A -85,B 0,C 180,E1 -10424.121,E2 -10424.121} C_VEL
LIN {X 0,Y 410.95,Z 881.619,A -85,B 0,C 180,E1 -10426.147,E2 -10426.147} C_VEL
LIN {X 0,Y 411.016,Z 881.98,A -85,B 0,C 180,E1 -10427.156,E2 -10427.156} C_VEL
LIN {X 0,Y 411.018,Z 881.878,A -85,B 0,C 180,E1 -10428.159,E2 -10428.159} C_VEL
LIN {X 0,Y 411.222,Z 880.438,A -85,B 0,C 180,E1 -10430.159,E2 -10430.159} C_VEL
LIN {X 0,Y 411.53,Z 877.154,A -85,B 0,C 180,E1 -10432.147,E2 -10432.147} C_VEL
LIN {X 0,Y 411.757,Z 874.957,A -85,B 0,C 180,E1 -10433.138,E2 -10433.138} C_VEL
LIN {X 0,Y 412.101,Z 870.592,A -85,B 0,C 180,E1 -10434.618,E2 -10434.618} C_VEL
LIN {X 0,Y 412.502,Z 864.978,A -85,B 0,C 180,E1 -10436.092,E2 -10436.092} C_VEL
LIN {X 0,Y 412.965,Z 859.245,A -85,B 0,C 180,E1 -10437.317,E2 -10437.317} C_VEL
LIN {X 0,Y 413.534,Z 852.297,A -85,B 0,C 180,E1 -10438.539,E2 -10438.539} C_VEL
LIN {X 0,Y 414.112,Z 843.873,A -85,B 0,C 180,E1 -10439.757,E2 -10439.757} C_VEL
LIN {X 0,Y 414.587,Z 836.519,A -85,B 0,C 180,E1 -10440.649,E2 -10440.649} C_VEL
LIN {X 0,Y 415.196,Z 827.48,A -85,B 0,C 180,E1 -10441.558,E2 -10441.558} C_VEL
LIN {X 0,Y 415.587,Z 818.658,A -85,B 0,C 180,E1 -10442.302,E2 -10442.302} C_VEL
LIN {X 0,Y 415.962,Z 808.363,A -85,B 0,C 180,E1 -10443.002,E2 -10443.002} C_VEL
LIN {X 0,Y 416.289,Z 797.895,A -85,B 0,C 180,E1 -10443.554,E2 -10443.554} C_VEL
LIN {X 0,Y 416.469,Z 787.246,A -85,B 0,C 180,E1 -10443.973,E2 -10443.973} C_VEL
LIN {X 0,Y 416.494,Z 774.095,A -85,B 0,C 180,E1 -10444.322,E2 -10444.322} C_VEL
LIN {X 0,Y 417.549,Z 716.874,A -85,B 0,C 180,E1 -10445.494,E2 -10445.494} C_VEL
LIN {X 0,Y 412.15,Z 703.521,A -85,B 0,C 180,E1 -10446.128,E2 -10446.128} C_VEL
LIN {X 0,Y 411.561,Z 701.867,A -85,B 0,C 180,E1 -10446.25,E2 -10446.25} C_VEL
LIN {X 0,Y 411.438,Z 701.267,A -85,B 0,C 180,E1 -10446.498,E2 -10446.498} C_VEL
LIN {X 0,Y 411.298,Z 701.252,A -85,B 0,C 180,E1 -10449.839,E2 -10449.839} C_VEL
LIN {X 0,Y 411.313,Z 701.248,A -85,B 0,C 180,E1 -10453.104,E2 -10453.104} C_VEL
LIN {X 0,Y 411.265,Z 701.257,A -85,B 0,C 180,E1 -10456.888,E2 -10456.888} C_VEL
LIN {X 0,Y 411.238,Z 701.26,A -85,B 0,C 180,E1 -10459.986,E2 -10459.986} C_VEL
LIN {X 0,Y 411.203,Z 701.262,A -85,B 0,C 180,E1 -10463.147,E2 -10463.147} C_VEL
LIN {X 0,Y 411.21,Z 701.265,A -85,B 0,C 180,E1 -10466.383,E2 -10466.383} C_VEL
LIN {X 0,Y 411.205,Z 701.262,A -85,B 0,C 180,E1 -10469.712,E2 -10469.712} C_VEL
LIN {X 0,Y 411.213,Z 701.265,A -85,B 0,C 180,E1 -10473.155,E2 -10473.155} C_VEL
LIN {X 0,Y 411.199,Z 701.264,A -85,B 0,C 180,E1 -10476.552,E2 -10476.552} C_VEL
LIN {X 0,Y 411.222,Z 701.261,A -85,B 0,C 180,E1 -10479.727,E2 -10479.727} C_VEL
LIN {X 0,Y 411.18,Z 701.267,A -85,B 0,C 180,E1 -10483.133,E2 -10483.133} C_VEL
LIN {X 0,Y 411.174,Z 701.268,A -85,B 0,C 180,E1 -10485.88,E2 -10485.88} C_VEL
LIN {X 0,Y 411.17,Z 701.267,A -85,B 0,C 180,E1 -10488.771,E2 -10488.771} C_VEL
LIN {X 0,Y 411.195,Z 701.264,A -85,B 0,C 180,E1 -10492.025,E2 -10492.025} C_VEL
LIN {X 0,Y 411.21,Z 701.263,A -85,B 0,C 180,E1 -10495.665,E2 -10495.665} C_VEL
LIN {X 0,Y 411.246,Z 701.477,A -85,B 0,C 180,E1 -10497.034,E2 -10497.034} C_VEL
LIN {X 0,Y 415.096,Z 717.75,A -85,B 0,C 180,E1 -10499.963,E2 -10499.963} C_VEL
LIN {X 0,Y 416.638,Z 725.574,A -85,B 0,C 180,E1 -10501.301,E2 -10501.301} C_VEL
LIN {X 0,Y 415.337,Z 744.182,A -85,B 0,C 180,E1 -10504.167,E2 -10504.167} C_VEL
LIN {X 0,Y 413.998,Z 764.651,A -85,B 0,C 180,E1 -10507.28,E2 -10507.28} C_VEL
LIN {X 0,Y 412.835,Z 787.043,A -85,B 0,C 180,E1 -10510.609,E2 -10510.609} C_VEL
LIN {X 0,Y 416.602,Z 823.702,A -85,B 0,C 180,E1 -10511.455,E2 -10511.455} C_VEL
LIN {X 0,Y 415.757,Z 897.308,A -85,B 0,C 180,E1 -10512.76,E2 -10512.76} C_VEL
LIN {X 0,Y 415.231,Z 910.641,A -85,B 0,C 180,E1 -10513.181,E2 -10513.181} C_VEL
LIN {X 0,Y 414.368,Z 923.992,A -85,B 0,C 180,E1 -10513.81,E2 -10513.81} C_VEL
LIN {X 0,Y 413.606,Z 936.06,A -85,B 0,C 180,E1 -10514.602,E2 -10514.602} C_VEL
LIN {X 0,Y 412.857,Z 946.325,A -85,B 0,C 180,E1 -10515.457,E2 -10515.457} C_VEL
LIN {X 0,Y 412.132,Z 956.912,A -85,B 0,C 180,E1 -10516.551,E2 -10516.551} C_VEL
LIN {X 0,Y 411.732,Z 963.984,A -85,B 0,C 180,E1 -10517.428,E2 -10517.428} C_VEL
LIN {X 0,Y 411.145,Z 972.373,A -85,B 0,C 180,E1 -10518.662,E2 -10518.662} C_VEL
LIN {X 0,Y 410.74,Z 980.629,A -85,B 0,C 180,E1 -10520.146,E2 -10520.146} C_VEL
LIN {X 0,Y 410.531,Z 987.289,A -85,B 0,C 180,E1 -10521.632,E2 -10521.632} C_VEL
LIN {X 0,Y 410.418,Z 993.178,A -85,B 0,C 180,E1 -10523.312,E2 -10523.312} C_VEL
LIN {X 0,Y 410.533,Z 997.817,A -85,B 0,C 180,E1 -10525.088,E2 -10525.088} C_VEL
LIN {X 0,Y 410.591,Z 999.753,A -85,B 0,C 180,E1 -10526.073,E2 -10526.073} C_VEL
LIN {X 0,Y 410.536,Z 1001.192,A -85,B 0,C 180,E1 -10527.055,E2 -10527.055} C_VEL
LIN {X 0,Y 410.553,Z 1002.215,A -85,B 0,C 180,E1 -10528.037,E2 -10528.037} C_VEL
LIN {X 0,Y 410.575,Z 1002.831,A -85,B 0,C 180,E1 -10529.018,E2 -10529.018} C_VEL
LIN {X 0,Y 410.597,Z 1003.044,A -85,B 0,C 180,E1 -10529.999,E2 -10529.999} C_VEL
LIN {X 0,Y 410.578,Z 1002.804,A -85,B 0,C 180,E1 -10530.979,E2 -10530.979} C_VEL
LIN {X 0,Y 410.56,Z 1002.15,A -85,B 0,C 180,E1 -10531.96,E2 -10531.96} C_VEL
LIN {X 0,Y 410.542,Z 1001.091,A -85,B 0,C 180,E1 -10532.942,E2 -10532.942} C_VEL
LIN {X 0,Y 410.593,Z 999.627,A -85,B 0,C 180,E1 -10533.924,E2 -10533.924} C_VEL
LIN {X 0,Y 410.462,Z 996.526,A -85,B 0,C 180,E1 -10535.402,E2 -10535.402} C_VEL
LIN {X 0,Y 410.431,Z 992.366,A -85,B 0,C 180,E1 -10536.883,E2 -10536.883} C_VEL
LIN {X 0,Y 410.557,Z 986.012,A -85,B 0,C 180,E1 -10538.613,E2 -10538.613} C_VEL
LIN {X 0,Y 410.755,Z 979.092,A -85,B 0,C 180,E1 -10540.099,E2 -10540.099} C_VEL
LIN {X 0,Y 411.231,Z 970.567,A -85,B 0,C 180,E1 -10541.583,E2 -10541.583} C_VEL
LIN {X 0,Y 411.902,Z 961.89,A -85,B 0,C 180,E1 -10542.814,E2 -10542.814} C_VEL
LIN {X 0,Y 412.464,Z 952.383,A -85,B 0,C 180,E1 -10543.925,E2 -10543.925} C_VEL
LIN {X 0,Y 413.102,Z 942.094,A -85,B 0,C 180,E1 -10544.909,E2 -10544.909} C_VEL
LIN {X 0,Y 413.98,Z 930.958,A -85,B 0,C 180,E1 -10545.759,E2 -10545.759} C_VEL
LIN {X 0,Y 414.701,Z 918.654,A -85,B 0,C 180,E1 -10546.489,E2 -10546.489} C_VEL
LIN {X 0,Y 415.439,Z 905.901,A -85,B 0,C 180,E1 -10547.029,E2 -10547.029} C_VEL
LIN {X 0,Y 415.88,Z 892.573,A -85,B 0,C 180,E1 -10547.39,E2 -10547.39} C_VEL
LIN {X 0,Y 416.659,Z 821.624,A -85,B 0,C 180,E1 -10548.639,E2 -10548.639} C_VEL
LIN {X 0,Y 412.77,Z 785.661,A -85,B 0,C 180,E1 -10549.486,E2 -10549.486} C_VEL
LIN {X 0,Y 412.831,Z 782.481,A -85,B 0,C 180,E1 -10549.904,E2 -10549.904} C_VEL
LIN {X 0,Y 414.211,Z 759.646,A -85,B 0,C 180,E1 -10553.343,E2 -10553.343} C_VEL
LIN {X 0,Y 415.86,Z 734.869,A -85,B 0,C 180,E1 -10557.147,E2 -10557.147} C_VEL
LIN {X 0,Y 416.507,Z 725.142,A -85,B 0,C 180,E1 -10558.666,E2 -10558.666} C_VEL
LIN {X 0,Y 413.863,Z 712.461,A -85,B 0,C 180,E1 -10560.891,E2 -10560.891} C_VEL
LIN {X 0,Y 411.23,Z 701.366,A -85,B 0,C 180,E1 -10562.988,E2 -10562.988} C_VEL
LIN {X 0,Y 411.192,Z 701.267,A -85,B 0,C 180,E1 -10565.527,E2 -10565.527} C_VEL
LIN {X 0,Y 411.21,Z 701.263,A -85,B 0,C 180,E1 -10569.223,E2 -10569.223} C_VEL
LIN {X 0,Y 411.174,Z 701.265,A -85,B 0,C 180,E1 -10572.695,E2 -10572.695} C_VEL
LIN {X 0,Y 411.165,Z 701.263,A -85,B 0,C 180,E1 -10575.879,E2 -10575.879} C_VEL
LIN {X 0,Y 411.157,Z 701.269,A -85,B 0,C 180,E1 -10578.77,E2 -10578.77} C_VEL
LIN {X 0,Y 411.191,Z 701.263,A -85,B 0,C 180,E1 -10582.026,E2 -10582.026} C_VEL
LIN {X 0,Y 411.197,Z 701.261,A -85,B 0,C 180,E1 -10585.666,E2 -10585.666} C_VEL
LIN {X 0,Y 411.187,Z 701.265,A -85,B 0,C 180,E1 -10589.152,E2 -10589.152} C_VEL
LIN {X 0,Y 411.249,Z 701.253,A -85,B 0,C 180,E1 -10592.522,E2 -10592.522} C_VEL
LIN {X 0,Y 411.216,Z 701.263,A -85,B 0,C 180,E1 -10595.784,E2 -10595.784} C_VEL
LIN {X 0,Y 411.185,Z 701.259,A -85,B 0,C 180,E1 -10598.965,E2 -10598.965} C_VEL
LIN {X 0,Y 411.241,Z 701.253,A -85,B 0,C 180,E1 -10602.085,E2 -10602.085} C_VEL
LIN {X 0,Y 411.252,Z 701.255,A -85,B 0,C 180,E1 -10605.147,E2 -10605.147} C_VEL
LIN {X 0,Y 411.272,Z 701.257,A -85,B 0,C 180,E1 -10608.167,E2 -10608.167} C_VEL
LIN {X 0,Y 411.428,Z 701.234,A -85,B 0,C 180,E1 -10612.189,E2 -10612.189} C_VEL
LIN {X 0,Y 411.459,Z 701.233,A -85,B 0,C 180,E1 -10614.118,E2 -10614.118} C_VEL
LIN {X 0,Y 411.502,Z 701.227,A -85,B 0,C 180,E1 -10618.043,E2 -10618.043} C_VEL
LIN {X 0,Y 411.629,Z 701.207,A -85,B 0,C 180,E1 -10620,E2 -10620} C_VEL
LIN {X 0,Y 411.453,Z 701.229,A -85,B 0,C 180,E1 -10622.937,E2 -10622.937} C_VEL
LIN {X 0,Y 411.446,Z 701.233,A -85,B 0,C 180,E1 -10626.867,E2 -10626.867} C_VEL
LIN {X 0,Y 411.343,Z 701.243,A -85,B 0,C 180,E1 -10628.846,E2 -10628.846} C_VEL
LIN {X 0,Y 411.273,Z 701.25,A -85,B 0,C 180,E1 -10631.833,E2 -10631.833} C_VEL
LIN {X 0,Y 411.248,Z 701.26,A -85,B 0,C 180,E1 -10634.853,E2 -10634.853} C_VEL
LIN {X 0,Y 411.239,Z 701.256,A -85,B 0,C 180,E1 -10637.916,E2 -10637.916} C_VEL
LIN {X 0,Y 411.185,Z 701.269,A -85,B 0,C 180,E1 -10641.035,E2 -10641.035} C_VEL
LIN {X 0,Y 411.2,Z 701.253,A -85,B 0,C 180,E1 -10644.217,E2 -10644.217} C_VEL
LIN {X 0,Y 411.248,Z 701.253,A -85,B 0,C 180,E1 -10647.479,E2 -10647.479} C_VEL
LIN {X 0,Y 411.18,Z 701.268,A -85,B 0,C 180,E1 -10650.849,E2 -10650.849} C_VEL
LIN {X 0,Y 411.197,Z 701.264,A -85,B 0,C 180,E1 -10654.335,E2 -10654.335} C_VEL
LIN {X 0,Y 411.193,Z 701.263,A -85,B 0,C 180,E1 -10657.974,E2 -10657.974} C_VEL
LIN {X 0,Y 411.176,Z 701.266,A -85,B 0,C 180,E1 -10660.505,E2 -10660.505} C_VEL
LIN {X 0,Y 411.166,Z 701.266,A -85,B 0,C 180,E1 -10663.135,E2 -10663.135} C_VEL
LIN {X 0,Y 411.209,Z 701.383,A -85,B 0,C 180,E1 -10665.764,E2 -10665.764} C_VEL
LIN {X 0,Y 411.453,Z 702.412,A -85,B 0,C 180,E1 -10665.957,E2 -10665.957} C_VEL
LIN {X 0,Y 417.612,Z 717.803,A -85,B 0,C 180,E1 -10666.576,E2 -10666.576} C_VEL
LIN {X 0,Y 416.999,Z 782.037,A -85,B 0,C 180,E1 -10667.735,E2 -10667.735} C_VEL
LIN {X 0,Y 416.886,Z 795.014,A -85,B 0,C 180,E1 -10668.139,E2 -10668.139} C_VEL
LIN {X 0,Y 416.645,Z 808.459,A -85,B 0,C 180,E1 -10668.787,E2 -10668.787} C_VEL
LIN {X 0,Y 416.236,Z 820.404,A -85,B 0,C 180,E1 -10669.571,E2 -10669.571} C_VEL
LIN {X 0,Y 415.626,Z 831.254,A -85,B 0,C 180,E1 -10670.492,E2 -10670.492} C_VEL
LIN {X 0,Y 414.937,Z 842.177,A -85,B 0,C 180,E1 -10671.661,E2 -10671.661} C_VEL
LIN {X 0,Y 414.218,Z 851.412,A -85,B 0,C 180,E1 -10672.888,E2 -10672.888} C_VEL
LIN {X 0,Y 413.583,Z 858.926,A -85,B 0,C 180,E1 -10674.11,E2 -10674.11} C_VEL
LIN {X 0,Y 413.017,Z 866.082,A -85,B 0,C 180,E1 -10675.545,E2 -10675.545} C_VEL
LIN {X 0,Y 412.468,Z 871.795,A -85,B 0,C 180,E1 -10676.961,E2 -10676.961} C_VEL
LIN {X 0,Y 412.009,Z 876.765,A -85,B 0,C 180,E1 -10678.529,E2 -10678.529} C_VEL
LIN {X 0,Y 411.666,Z 880.96,A -85,B 0,C 180,E1 -10680.326,E2 -10680.326} C_VEL
LIN {X 0,Y 411.466,Z 882.774,A -85,B 0,C 180,E1 -10681.431,E2 -10681.431} C_VEL
LIN {X 0,Y 411.355,Z 884.235,A -85,B 0,C 180,E1 -10682.676,E2 -10682.676} C_VEL
LIN {X 0,Y 411.272,Z 884.889,A -85,B 0,C 180,E1 -10683.623,E2 -10683.623} C_VEL
LIN {X 0,Y 411.193,Z 885.228,A -85,B 0,C 180,E1 -10684.941,E2 -10684.941} C_VEL
LIN {X 0,Y 411.194,Z 884.438,A -85,B 0,C 180,E1 -10686.854,E2 -10686.854} C_VEL
LIN {X 0,Y 411.277,Z 883.36,A -85,B 0,C 180,E1 -10687.919,E2 -10687.919} C_VEL
LIN {X 0,Y 411.438,Z 881.823,A -85,B 0,C 180,E1 -10688.981,E2 -10688.981} C_VEL
LIN {X 0,Y 411.717,Z 878.597,A -85,B 0,C 180,E1 -10690.559,E2 -10690.559} C_VEL
LIN {X 0,Y 412.083,Z 874.226,A -85,B 0,C 180,E1 -10692.124,E2 -10692.124} C_VEL
LIN {X 0,Y 412.49,Z 868.62,A -85,B 0,C 180,E1 -10693.674,E2 -10693.674} C_VEL
LIN {X 0,Y 413.034,Z 861.579,A -85,B 0,C 180,E1 -10695.214,E2 -10695.214} C_VEL
LIN {X 0,Y 413.652,Z 854.335,A -85,B 0,C 180,E1 -10696.492,E2 -10696.492} C_VEL
LIN {X 0,Y 414.249,Z 845.597,A -85,B 0,C 180,E1 -10697.758,E2 -10697.758} C_VEL
LIN {X 0,Y 414.893,Z 835.617,A -85,B 0,C 180,E1 -10698.929,E2 -10698.929} C_VEL
LIN {X 0,Y 415.471,Z 825.343,A -85,B 0,C 180,E1 -10699.905,E2 -10699.905} C_VEL
LIN {X 0,Y 416.039,Z 813.93,A -85,B 0,C 180,E1 -10700.767,E2 -10700.767} C_VEL
LIN {X 0,Y 416.38,Z 802.124,A -85,B 0,C 180,E1 -10701.447,E2 -10701.447} C_VEL
LIN {X 0,Y 416.561,Z 788.698,A -85,B 0,C 180,E1 -10702.001,E2 -10702.001} C_VEL
LIN {X 0,Y 416.635,Z 776.85,A -85,B 0,C 180,E1 -10702.307,E2 -10702.307} C_VEL
LIN {X 0,Y 416.764,Z 754.865,A -85,B 0,C 180,E1 -10702.698,E2 -10702.698} C_VEL
LIN {X 0,Y 416.154,Z 749.058,A -85,B 0,C 180,E1 -10702.831,E2 -10702.831} C_VEL
LIN {X 0,Y 410.914,Z 730.38,A -85,B 0,C 180,E1 -10703.411,E2 -10703.411} C_VEL
LIN {X 0,Y 410.43,Z 724.572,A -85,B 0,C 180,E1 -10703.541,E2 -10703.541} C_VEL
LIN {X 0,Y 410.328,Z 718.117,A -85,B 0,C 180,E1 -10703.665,E2 -10703.665} C_VEL
LIN {X 0,Y 404.596,Z 703.107,A -85,B 0,C 180,E1 -10704.238,E2 -10704.238} C_VEL
LIN {X 0,Y 404.362,Z 702.227,A -85,B 0,C 180,E1 -10704.422,E2 -10704.422} C_VEL
LIN {X 0,Y 404.474,Z 702.102,A -85,B 0,C 180,E1 -10708.01,E2 -10708.01} C_VEL
LIN {X 0,Y 404.352,Z 702.117,A -85,B 0,C 180,E1 -10710.997,E2 -10710.997} C_VEL
LIN {X 0,Y 404.362,Z 702.116,A -85,B 0,C 180,E1 -10712.99,E2 -10712.99} C_VEL
LIN {X 0,Y 404.371,Z 702.117,A -85,B 0,C 180,E1 -10715.987,E2 -10715.987} C_VEL
LIN {X 0,Y 404.259,Z 702.128,A -85,B 0,C 180,E1 -10719.003,E2 -10719.003} C_VEL
LIN {X 0,Y 404.252,Z 702.126,A -85,B 0,C 180,E1 -10722.043,E2 -10722.043} C_VEL
LIN {X 0,Y 404.204,Z 702.13,A -85,B 0,C 180,E1 -10725.119,E2 -10725.119} C_VEL
LIN {X 0,Y 404.193,Z 702.135,A -85,B 0,C 180,E1 -10728.24,E2 -10728.24} C_VEL
LIN {X 0,Y 404.139,Z 702.141,A -85,B 0,C 180,E1 -10731.421,E2 -10731.421} C_VEL
LIN {X 0,Y 404.141,Z 702.143,A -85,B 0,C 180,E1 -10734.669,E2 -10734.669} C_VEL
LIN {X 0,Y 404.104,Z 702.138,A -85,B 0,C 180,E1 -10738.008,E2 -10738.008} C_VEL
LIN {X 0,Y 404.145,Z 702.14,A -85,B 0,C 180,E1 -10740.287,E2 -10740.287} C_VEL
LIN {X 0,Y 404.142,Z 702.124,A -85,B 0,C 180,E1 -10743.814,E2 -10743.814} C_VEL
LIN {X 0,Y 404.136,Z 702.131,A -85,B 0,C 180,E1 -10746.874,E2 -10746.874} C_VEL
LIN {X 0,Y 404.124,Z 702.143,A -85,B 0,C 180,E1 -10750.075,E2 -10750.075} C_VEL
LIN {X 0,Y 404.084,Z 702.149,A -85,B 0,C 180,E1 -10753.073,E2 -10753.073} C_VEL
LIN {X 0,Y 404.124,Z 702.147,A -85,B 0,C 180,E1 -10755.922,E2 -10755.922} C_VEL
LIN {X 0,Y 404.107,Z 702.145,A -85,B 0,C 180,E1 -10758.633,E2 -10758.633} C_VEL
LIN {X 0,Y 404.139,Z 702.145,A -85,B 0,C 180,E1 -10761.497,E2 -10761.497} C_VEL
LIN {X 0,Y 404.166,Z 702.139,A -85,B 0,C 180,E1 -10764.982,E2 -10764.982} C_VEL
LIN {X 0,Y 404.191,Z 702.333,A -85,B 0,C 180,E1 -10768.147,E2 -10768.147} C_VEL
LIN {X 0,Y 404.459,Z 703.486,A -85,B 0,C 180,E1 -10768.315,E2 -10768.315} C_VEL
LIN {X 0,Y 409.547,Z 717.729,A -85,B 0,C 180,E1 -10768.83,E2 -10768.83} C_VEL
LIN {X 0,Y 408.676,Z 778.797,A -85,B 0,C 180,E1 -10770.059,E2 -10770.059} C_VEL
LIN {X 0,Y 408.481,Z 789.909,A -85,B 0,C 180,E1 -10770.424,E2 -10770.424} C_VEL
LIN {X 0,Y 408.223,Z 800.269,A -85,B 0,C 180,E1 -10770.898,E2 -10770.898} C_VEL
LIN {X 0,Y 407.951,Z 810.05,A -85,B 0,C 180,E1 -10771.477,E2 -10771.477} C_VEL
LIN {X 0,Y 407.465,Z 820.413,A -85,B 0,C 180,E1 -10772.244,E2 -10772.244} C_VEL
LIN {X 0,Y 407.063,Z 829.318,A -85,B 0,C 180,E1 -10773.05,E2 -10773.05} C_VEL
LIN {X 0,Y 406.508,Z 838.346,A -85,B 0,C 180,E1 -10774.031,E2 -10774.031} C_VEL
LIN {X 0,Y 406.05,Z 847.089,A -85,B 0,C 180,E1 -10775.182,E2 -10775.182} C_VEL
LIN {X 0,Y 405.626,Z 853.907,A -85,B 0,C 180,E1 -10776.244,E2 -10776.244} C_VEL
LIN {X 0,Y 405.12,Z 860.981,A -85,B 0,C 180,E1 -10777.564,E2 -10777.564} C_VEL
LIN {X 0,Y 404.734,Z 866.801,A -85,B 0,C 180,E1 -10778.88,E2 -10778.88} C_VEL
LIN {X 0,Y 404.508,Z 871.637,A -85,B 0,C 180,E1 -10780.221,E2 -10780.221} C_VEL
LIN {X 0,Y 404.325,Z 874.764,A -85,B 0,C 180,E1 -10781.242,E2 -10781.242} C_VEL
LIN {X 0,Y 404.092,Z 878.84,A -85,B 0,C 180,E1 -10783.055,E2 -10783.055} C_VEL
LIN {X 0,Y 404.003,Z 880.199,A -85,B 0,C 180,E1 -10783.839,E2 -10783.839} C_VEL
LIN {X 0,Y 403.929,Z 882.502,A -85,B 0,C 180,E1 -10785.901,E2 -10785.901} C_VEL
LIN {X 0,Y 403.958,Z 882.988,A -85,B 0,C 180,E1 -10786.982,E2 -10786.982} C_VEL
LIN {X 0,Y 404.001,Z 883.034,A -85,B 0,C 180,E1 -10787.951,E2 -10787.951} C_VEL
LIN {X 0,Y 404.201,Z 881.77,A -85,B 0,C 180,E1 -10789.987,E2 -10789.987} C_VEL
LIN {X 0,Y 404.549,Z 878.805,A -85,B 0,C 180,E1 -10792.011,E2 -10792.011} C_VEL
LIN {X 0,Y 404.862,Z 875.382,A -85,B 0,C 180,E1 -10793.521,E2 -10793.521} C_VEL
LIN {X 0,Y 405.245,Z 870.825,A -85,B 0,C 180,E1 -10795.025,E2 -10795.025} C_VEL
LIN {X 0,Y 405.617,Z 866.111,A -85,B 0,C 180,E1 -10796.274,E2 -10796.274} C_VEL
LIN {X 0,Y 406.124,Z 860.368,A -85,B 0,C 180,E1 -10797.52,E2 -10797.52} C_VEL
LIN {X 0,Y 406.719,Z 853.421,A -85,B 0,C 180,E1 -10798.762,E2 -10798.762} C_VEL
LIN {X 0,Y 407.341,Z 845.024,A -85,B 0,C 180,E1 -10800,E2 -10800} C_VEL
LIN {X 0,Y 407.891,Z 836.962,A -85,B 0,C 180,E1 -10800.987,E2 -10800.987} C_VEL
LIN {X 0,Y 408.478,Z 828.705,A -85,B 0,C 180,E1 -10801.831,E2 -10801.831} C_VEL
LIN {X 0,Y 408.902,Z 819.922,A -85,B 0,C 180,E1 -10802.586,E2 -10802.586} C_VEL
LIN {X 0,Y 409.306,Z 809.223,A -85,B 0,C 180,E1 -10803.322,E2 -10803.322} C_VEL
LIN {X 0,Y 409.647,Z 798.875,A -85,B 0,C 180,E1 -10803.873,E2 -10803.873} C_VEL
LIN {X 0,Y 409.847,Z 788.985,A -85,B 0,C 180,E1 -10804.272,E2 -10804.272} C_VEL
LIN {X 0,Y 409.863,Z 777.005,A -85,B 0,C 180,E1 -10804.611,E2 -10804.611} C_VEL
LIN {X 0,Y 410.949,Z 718.457,A -85,B 0,C 180,E1 -10805.851,E2 -10805.851} C_VEL
LIN {X 0,Y 405.585,Z 705.28,A -85,B 0,C 180,E1 -10806.505,E2 -10806.505} C_VEL
LIN {X 0,Y 404.541,Z 702.865,A -85,B 0,C 180,E1 -10806.671,E2 -10806.671} C_VEL
LIN {X 0,Y 404.413,Z 702.185,A -85,B 0,C 180,E1 -10806.862,E2 -10806.862} C_VEL
LIN {X 0,Y 404.264,Z 702.128,A -85,B 0,C 180,E1 -10810.011,E2 -10810.011} C_VEL
LIN {X 0,Y 404.274,Z 702.125,A -85,B 0,C 180,E1 -10813.211,E2 -10813.211} C_VEL
LIN {X 0,Y 404.223,Z 702.134,A -85,B 0,C 180,E1 -10817.007,E2 -10817.007} C_VEL
LIN {X 0,Y 404.171,Z 702.141,A -85,B 0,C 180,E1 -10820.351,E2 -10820.351} C_VEL
LIN {X 0,Y 404.168,Z 702.138,A -85,B 0,C 180,E1 -10823.575,E2 -10823.575} C_VEL
LIN {X 0,Y 404.158,Z 702.142,A -85,B 0,C 180,E1 -10826.88,E2 -10826.88} C_VEL
LIN {X 0,Y 404.151,Z 702.142,A -85,B 0,C 180,E1 -10830.285,E2 -10830.285} C_VEL
LIN {X 0,Y 404.151,Z 702.14,A -85,B 0,C 180,E1 -10833.812,E2 -10833.812} C_VEL
LIN {X 0,Y 404.143,Z 702.143,A -85,B 0,C 180,E1 -10836.874,E2 -10836.874} C_VEL
LIN {X 0,Y 404.154,Z 702.14,A -85,B 0,C 180,E1 -10840.079,E2 -10840.079} C_VEL
LIN {X 0,Y 404.159,Z 702.141,A -85,B 0,C 180,E1 -10843.083,E2 -10843.083} C_VEL
LIN {X 0,Y 404.154,Z 702.142,A -85,B 0,C 180,E1 -10845.925,E2 -10845.925} C_VEL
LIN {X 0,Y 404.124,Z 702.144,A -85,B 0,C 180,E1 -10848.634,E2 -10848.634} C_VEL
LIN {X 0,Y 404.154,Z 702.143,A -85,B 0,C 180,E1 -10851.492,E2 -10851.492} C_VEL
LIN {X 0,Y 404.189,Z 702.139,A -85,B 0,C 180,E1 -10854.983,E2 -10854.983} C_VEL
LIN {X 0,Y 404.207,Z 702.365,A -85,B 0,C 180,E1 -10856.719,E2 -10856.719} C_VEL
LIN {X 0,Y 408.302,Z 719.654,A -85,B 0,C 180,E1 -10859.891,E2 -10859.891} C_VEL
LIN {X 0,Y 409.771,Z 727.798,A -85,B 0,C 180,E1 -10861.298,E2 -10861.298} C_VEL
LIN {X 0,Y 408.148,Z 748.31,A -85,B 0,C 180,E1 -10864.5,E2 -10864.5} C_VEL
LIN {X 0,Y 406.9,Z 767.044,A -85,B 0,C 180,E1 -10867.398,E2 -10867.398} C_VEL
LIN {X 0,Y 405.877,Z 785.968,A -85,B 0,C 180,E1 -10870.265,E2 -10870.265} C_VEL
LIN {X 0,Y 409.806,Z 823.521,A -85,B 0,C 180,E1 -10871.163,E2 -10871.163} C_VEL
LIN {X 0,Y 408.891,Z 896.977,A -85,B 0,C 180,E1 -10872.494,E2 -10872.494} C_VEL
LIN {X 0,Y 408.327,Z 910.852,A -85,B 0,C 180,E1 -10872.953,E2 -10872.953} C_VEL
LIN {X 0,Y 407.449,Z 923.83,A -85,B 0,C 180,E1 -10873.592,E2 -10873.592} C_VEL
LIN {X 0,Y 406.602,Z 936.492,A -85,B 0,C 180,E1 -10874.458,E2 -10874.458} C_VEL
LIN {X 0,Y 405.833,Z 946.5,A -85,B 0,C 180,E1 -10875.328,E2 -10875.328} C_VEL
LIN {X 0,Y 405.066,Z 957.032,A -85,B 0,C 180,E1 -10876.456,E2 -10876.456} C_VEL
LIN {X 0,Y 404.578,Z 964.71,A -85,B 0,C 180,E1 -10877.457,E2 -10877.457} C_VEL
LIN {X 0,Y 404.048,Z 972.827,A -85,B 0,C 180,E1 -10878.714,E2 -10878.714} C_VEL
LIN {X 0,Y 403.623,Z 980.799,A -85,B 0,C 180,E1 -10880.224,E2 -10880.224} C_VEL
LIN {X 0,Y 403.402,Z 988.132,A -85,B 0,C 180,E1 -10881.987,E2 -10881.987} C_VEL
LIN {X 0,Y 403.348,Z 992.471,A -85,B 0,C 180,E1 -10883.304,E2 -10883.304} C_VEL
LIN {X 0,Y 403.463,Z 996.795,A -85,B 0,C 180,E1 -10885.002,E2 -10885.002} C_VEL
LIN {X 0,Y 403.556,Z 998.738,A -85,B 0,C 180,E1 -10886.004,E2 -10886.004} C_VEL
LIN {X 0,Y 403.496,Z 1000.181,A -85,B 0,C 180,E1 -10887.003,E2 -10887.003} C_VEL
LIN {X 0,Y 403.516,Z 1001.204,A -85,B 0,C 180,E1 -10888.002,E2 -10888.002} C_VEL
LIN {X 0,Y 403.543,Z 1001.822,A -85,B 0,C 180,E1 -10889.001,E2 -10889.001} C_VEL
LIN {X 0,Y 403.569,Z 1002.037,A -85,B 0,C 180,E1 -10889.999,E2 -10889.999} C_VEL
LIN {X 0,Y 403.546,Z 1001.798,A -85,B 0,C 180,E1 -10890.996,E2 -10890.996} C_VEL
LIN {X 0,Y 403.522,Z 1001.141,A -85,B 0,C 180,E1 -10891.995,E2 -10891.995} C_VEL
LIN {X 0,Y 403.559,Z 998.617,A -85,B 0,C 180,E1 -10893.993,E2 -10893.993} C_VEL
LIN {X 0,Y 403.388,Z 995.508,A -85,B 0,C 180,E1 -10895.497,E2 -10895.497} C_VEL
LIN {X 0,Y 403.386,Z 991.351,A -85,B 0,C 180,E1 -10897.004,E2 -10897.004} C_VEL
LIN {X 0,Y 403.495,Z 984.999,A -85,B 0,C 180,E1 -10898.765,E2 -10898.765} C_VEL
LIN {X 0,Y 403.703,Z 978.085,A -85,B 0,C 180,E1 -10900.277,E2 -10900.277} C_VEL
LIN {X 0,Y 404.191,Z 969.564,A -85,B 0,C 180,E1 -10901.787,E2 -10901.787} C_VEL
LIN {X 0,Y 404.941,Z 959.676,A -85,B 0,C 180,E1 -10903.195,E2 -10903.195} C_VEL
LIN {X 0,Y 405.656,Z 949.008,A -85,B 0,C 180,E1 -10904.42,E2 -10904.42} C_VEL
LIN {X 0,Y 406.291,Z 939.684,A -85,B 0,C 180,E1 -10905.294,E2 -10905.294} C_VEL
LIN {X 0,Y 407.2,Z 928.227,A -85,B 0,C 180,E1 -10906.158,E2 -10906.158} C_VEL
LIN {X 0,Y 407.995,Z 916.579,A -85,B 0,C 180,E1 -10906.833,E2 -10906.833} C_VEL
LIN {X 0,Y 408.752,Z 903.268,A -85,B 0,C 180,E1 -10907.38,E2 -10907.38} C_VEL
LIN {X 0,Y 409.122,Z 890.44,A -85,B 0,C 180,E1 -10907.719,E2 -10907.719} C_VEL
LIN {X 0,Y 409.927,Z 822.47,A -85,B 0,C 180,E1 -10908.932,E2 -10908.932} C_VEL
LIN {X 0,Y 406.009,Z 785.972,A -85,B 0,C 180,E1 -10909.812,E2 -10909.812} C_VEL
LIN {X 0,Y 405.803,Z 783.897,A -85,B 0,C 180,E1 -10909.9,E2 -10909.9} C_VEL
LIN {X 0,Y 407.213,Z 761.11,A -85,B 0,C 180,E1 -10913.386,E2 -10913.386} C_VEL
LIN {X 0,Y 408.994,Z 735.69,A -85,B 0,C 180,E1 -10917.363,E2 -10917.363} C_VEL
LIN {X 0,Y 409.694,Z 727.229,A -85,B 0,C 180,E1 -10918.704,E2 -10918.704} C_VEL
LIN {X 0,Y 407.427,Z 715.806,A -85,B 0,C 180,E1 -10920.737,E2 -10920.737} C_VEL
LIN {X 0,Y 404.17,Z 702.246,A -85,B 0,C 180,E1 -10923.341,E2 -10923.341} C_VEL
LIN {X 0,Y 404.135,Z 702.144,A -85,B 0,C 180,E1 -10926.245,E2 -10926.245} C_VEL
LIN {X 0,Y 404.147,Z 702.143,A -85,B 0,C 180,E1 -10928.756,E2 -10928.756} C_VEL
LIN {X 0,Y 404.115,Z 702.146,A -85,B 0,C 180,E1 -10931.598,E2 -10931.598} C_VEL
LIN {X 0,Y 404.139,Z 702.145,A -85,B 0,C 180,E1 -10934.521,E2 -10934.521} C_VEL
LIN {X 0,Y 404.131,Z 702.146,A -85,B 0,C 180,E1 -10937.295,E2 -10937.295} C_VEL
LIN {X 0,Y 404.16,Z 702.13,A -85,B 0,C 180,E1 -10939.954,E2 -10939.954} C_VEL
LIN {X 0,Y 404.13,Z 702.141,A -85,B 0,C 180,E1 -10943.123,E2 -10943.123} C_VEL
LIN {X 0,Y 404.135,Z 702.139,A -85,B 0,C 180,E1 -10946.187,E2 -10946.187} C_VEL
LIN {X 0,Y 404.143,Z 702.143,A -85,B 0,C 180,E1 -10949.715,E2 -10949.715} C_VEL
LIN {X 0,Y 404.185,Z 702.137,A -85,B 0,C 180,E1 -10953.122,E2 -10953.122} C_VEL
LIN {X 0,Y 404.166,Z 702.138,A -85,B 0,C 180,E1 -10955.334,E2 -10955.334} C_VEL
LIN {X 0,Y 404.127,Z 702.137,A -85,B 0,C 180,E1 -10958.58,E2 -10958.58} C_VEL
LIN {X 0,Y 404.199,Z 702.134,A -85,B 0,C 180,E1 -10961.761,E2 -10961.761} C_VEL
LIN {X 0,Y 404.199,Z 702.133,A -85,B 0,C 180,E1 -10964.882,E2 -10964.882} C_VEL
LIN {X 0,Y 404.244,Z 702.13,A -85,B 0,C 180,E1 -10967.958,E2 -10967.958} C_VEL
LIN {X 0,Y 404.392,Z 702.109,A -85,B 0,C 180,E1 -10972.129,E2 -10972.129} C_VEL
LIN {X 0,Y 404.407,Z 702.113,A -85,B 0,C 180,E1 -10974.015,E2 -10974.015} C_VEL
LIN {X 0,Y 404.471,Z 702.102,A -85,B 0,C 180,E1 -10978.009,E2 -10978.009} C_VEL
LIN {X 0,Y 404.599,Z 702.082,A -85,B 0,C 180,E1 -10980,E2 -10980} C_VEL
LIN {X 0,Y 404.41,Z 702.106,A -85,B 0,C 180,E1 -10982.989,E2 -10982.989} C_VEL
LIN {X 0,Y 404.398,Z 702.11,A -85,B 0,C 180,E1 -10986.988,E2 -10986.988} C_VEL
LIN {X 0,Y 404.248,Z 702.126,A -85,B 0,C 180,E1 -10990.012,E2 -10990.012} C_VEL
LIN {X 0,Y 404.255,Z 702.129,A -85,B 0,C 180,E1 -10993.212,E2 -10993.212} C_VEL
LIN {X 0,Y 404.204,Z 702.136,A -85,B 0,C 180,E1 -10997.008,E2 -10997.008} C_VEL
LIN {X 0,Y 404.152,Z 702.139,A -85,B 0,C 180,E1 -11000.352,E2 -11000.352} C_VEL
LIN {X 0,Y 404.149,Z 702.129,A -85,B 0,C 180,E1 -11003.576,E2 -11003.576} C_VEL
LIN {X 0,Y 404.17,Z 702.141,A -85,B 0,C 180,E1 -11005.768,E2 -11005.768} C_VEL
LIN {X 0,Y 404.184,Z 702.128,A -85,B 0,C 180,E1 -11008.001,E2 -11008.001} C_VEL
LIN {X 0,Y 404.13,Z 702.143,A -85,B 0,C 180,E1 -11011.559,E2 -11011.559} C_VEL
LIN {X 0,Y 404.177,Z 702.139,A -85,B 0,C 180,E1 -11015.017,E2 -11015.017} C_VEL
LIN {X 0,Y 404.151,Z 702.136,A -85,B 0,C 180,E1 -11018.758,E2 -11018.758} C_VEL
LIN {X 0,Y 404.116,Z 702.146,A -85,B 0,C 180,E1 -11021.601,E2 -11021.601} C_VEL
LIN {X 0,Y 404.121,Z 702.146,A -85,B 0,C 180,E1 -11024.959,E2 -11024.959} C_VEL
LIN {X 0,Y 404.208,Z 702.457,A -85,B 0,C 180,E1 -11025.469,E2 -11025.469} C_VEL
LIN {X 0,Y 404.548,Z 703.75,A -85,B 0,C 180,E1 -11025.614,E2 -11025.614} C_VEL
LIN {X 0,Y 411.002,Z 719.627,A -85,B 0,C 180,E1 -11026.27,E2 -11026.27} C_VEL
LIN {X 0,Y 410.284,Z 781.825,A -85,B 0,C 180,E1 -11027.404,E2 -11027.404} C_VEL
LIN {X 0,Y 410.216,Z 794.97,A -85,B 0,C 180,E1 -11027.8,E2 -11027.8} C_VEL
LIN {X 0,Y 410.014,Z 806.711,A -85,B 0,C 180,E1 -11028.344,E2 -11028.344} C_VEL
LIN {X 0,Y 409.645,Z 817.55,A -85,B 0,C 180,E1 -11029.015,E2 -11029.015} C_VEL
LIN {X 0,Y 409.055,Z 828.581,A -85,B 0,C 180,E1 -11029.89,E2 -11029.89} C_VEL
LIN {X 0,Y 408.419,Z 839.423,A -85,B 0,C 180,E1 -11030.978,E2 -11030.978} C_VEL
LIN {X 0,Y 407.673,Z 848.853,A -85,B 0,C 180,E1 -11032.152,E2 -11032.152} C_VEL
LIN {X 0,Y 406.958,Z 857.202,A -85,B 0,C 180,E1 -11033.432,E2 -11033.432} C_VEL
LIN {X 0,Y 406.329,Z 864.31,A -85,B 0,C 180,E1 -11034.764,E2 -11034.764} C_VEL
LIN {X 0,Y 405.725,Z 871.084,A -85,B 0,C 180,E1 -11036.339,E2 -11036.339} C_VEL
LIN {X 0,Y 405.207,Z 876.404,A -85,B 0,C 180,E1 -11037.912,E2 -11037.912} C_VEL
LIN {X 0,Y 404.78,Z 881.034,A -85,B 0,C 180,E1 -11039.769,E2 -11039.769} C_VEL
LIN {X 0,Y 404.537,Z 883.112,A -85,B 0,C 180,E1 -11040.895,E2 -11040.895} C_VEL
